			Cmd_RLen:=18;
			j:=(DelayAllarmeTemperaturaNonRaggiunta);   				(* Ritardo Allarme dall'avvio Caldaia*)
			TxLen:=TxLen+RAWTOHEX(ADR(j),2,ADR(TxData[TxLen]));
			j:=(DeltaInterventoAllarmeTempeaturaNonRaggiuta);			(* Delta Soglia Temperatura per Allarme Temperatura Non Raggiunta *)
			TxLen:=TxLen+RAWTOHEX(ADR(j),2,ADR(TxData[TxLen]));
			j:=(OffsetSetPointManuale);									(* Offest Perdite Scambiatore 1  *)
			TxLen:=TxLen+RAWTOHEX(ADR(j),2,ADR(TxData[TxLen]));
			j:=(OffsetSetPointManuale2);								(* Offest Perdite Scambiatore 2  *)
			TxLen:=TxLen+RAWTOHEX(ADR(j),2,ADR(TxData[TxLen]));
			j:=BOOL_TO_INT(BitAbilitaBoost);							(* Abilitazione controllo Boost  *)
			TxLen:=TxLen+RAWTOHEX(ADR(j),2,ADR(TxData[TxLen]));
			j:=BOOL_TO_INT(BitAbilitaBoost);										(* Offset al Setpoint della Caldaia per azione di Boost   *)
			TxLen:=TxLen+RAWTOHEX(ADR(j),2,ADR(TxData[TxLen]));




	6: (*  Scrivo i Parametri gestione Impianto - Antigelo   *)

			Cmd_Buf_U16:=ADR(Cmd_Buf[8]);
			SogliaMinStartAntigelo := Cmd_Buf_U16^; 			(* Soglia mininma Start Antigelo *)
			Cmd_Buf_U16:=ADR(Cmd_Buf[10]);
			SogliaMinStopAntigelo := Cmd_Buf_U16^;				(* Soglia Massima Stop Antigelo *)
			Cmd_Buf_U16:=ADR(Cmd_Buf[12]);
			BitAbilitaAntigelo :=INT_TO_BOOL( Cmd_Buf_U16^); 	(* Abilitazione Antigelo  *)

	7: (*  Leggi i parametri gestione Impianto - Antigelo *)

			Cmd_RLen:=14;
			j:=(SogliaMinStartAntigelo); 							(* Soglia mininma Start Antigelo *)
			TxLen:=TxLen+RAWTOHEX(ADR(j),2,ADR(TxData[TxLen]));
			j:=(SogliaMinStopAntigelo);								(* Soglia Massima Stop Antigelo *)
			TxLen:=TxLen+RAWTOHEX(ADR(j),2,ADR(TxData[TxLen]));
			j:=BOOL_TO_INT(BitAbilitaAntigelo);						(* Abilitazione Antigelo  *)
			TxLen:=TxLen+RAWTOHEX(ADR(j),2,ADR(TxData[TxLen]));

(*	10: (*  Scrivo i Parametri per la gestione della velocità dei circolatori sui primari   *)

			Cmd_Buf_U16:=ADR(Cmd_Buf[8]);
			PercVelMin := Cmd_Buf_U16^;
			Cmd_Buf_U16:=ADR(Cmd_Buf[10]);
			PercVelMax := Cmd_Buf_U16^;
			Cmd_Buf_U16:=ADR(Cmd_Buf[12]);
			ErroreTempMax := Cmd_Buf_U16^;
			Cmd_Buf_U16:=ADR(Cmd_Buf[14]);
			ErroreTempMin := Cmd_Buf_U16^;

	11: (*  Leggo i Parametri per la gestione della velocità dei circolatori sui primari   *)

			Cmd_RLen:=8;
			j:=(PercVelMin);
			TxLen:=TxLen+RAWTOHEX(ADR(j),2,ADR(TxData[TxLen]));
			j:=(PercVelMax);
			TxLen:=TxLen+RAWTOHEX(ADR(j),2,ADR(TxData[TxLen]));
			j:=(ErroreTempMax);
			TxLen:=TxLen+RAWTOHEX(ADR(j),2,ADR(TxData[TxLen]));
			j:=(ErroreTempMin);
			TxLen:=TxLen+RAWTOHEX(ADR(j),2,ADR(TxData[TxLen]));


	12: (*  Scrivo i Parametri per la gestione della velocità dei circolatori sui primari   *)


				Cmd_Buf_U16:=ADR(Cmd_Buf[8]);
				CAS01.DeltaTempThr := Cmd_Buf_U16^;
				Cmd_Buf_U16:=ADR(Cmd_Buf[10]);
				CAS01.Tmonitor_Off := DWORD_TO_TIME((Cmd_Buf_U16^)*60*1000);
				Cmd_Buf_U16:=ADR(Cmd_Buf[12]);
				CAS01.Tmonitor_On := DWORD_TO_TIME((Cmd_Buf_U16^)*60*1000);

	13: (*  Leggo i Parametri per la gestione della velocità dei circolatori sui primari   *)


				Cmd_RLen:=6;
				j:=(CAS01.DeltaTempThr);
				TxLen:=TxLen+RAWTOHEX(ADR(j),2,ADR(TxData[TxLen]));
				j:=DWORD_TO_WORD(TIME_TO_DWORD((CAS01.Tmonitor_Off)/60/1000));
				TxLen:=TxLen+RAWTOHEX(ADR(j),2,ADR(TxData[TxLen]));
				j:=DWORD_TO_WORD(TIME_TO_DWORD((CAS01.Tmonitor_On)/60/1000));
				TxLen:=TxLen+RAWTOHEX(ADR(j),2,ADR(TxData[TxLen]));


*)


	14: (*  Imposto data e ora del PLC  *)


			Cmd_Buf_U16:=ADR(Cmd_Buf[8]);
			SetAnno:= Cmd_Buf_U16^; 												(* Anno *)
			Cmd_Buf_U16:=ADR(Cmd_Buf[10]);
			SetMese:= Cmd_Buf_U16^;												 	(* mese *)
			Cmd_Buf_U16:=ADR(Cmd_Buf[12]);
			SetGiorno:=( Cmd_Buf_U16^);											 	(* Giorno *)
			Cmd_Buf_U16:=ADR(Cmd_Buf[14]);
			SetOra:=( Cmd_Buf_U16^); 												(* ora *)
			Cmd_Buf_U16:=ADR(Cmd_Buf[16]);
			SetMinuti:= ( Cmd_Buf_U16^);										 	(* Minuti *)
			Cmd_Buf_U16:=ADR(Cmd_Buf[18]);
			SetSecondi:= ( Cmd_Buf_U16^);										 	(* secondi *)

	(*		SysRtcSetTime(SetDataTime(DWORD_TO_INT(ADR(Cmd_Buf[8])),				(* Anno *)
										DWORD_TO_INT(ADR(Cmd_Buf[10])),				(* mese *)
										DWORD_TO_INT(ADR(Cmd_Buf[11])),				(* Giorno *)
										DWORD_TO_INT(ADR(Cmd_Buf[12])),				(* ora *)
										DWORD_TO_INT(ADR(Cmd_Buf[13])),				(* Minuti *)
										DWORD_TO_INT(ADR(Cmd_Buf[14]))				(* secondi *)
										)); *)

		SysRtcSetTime((SetDataTime(SetAnno,SetMese,SetGiorno,SetOra,SetMinuti,SetSecondi)));


ELSE
	Cmd_R:=3;
END_CASE
END_ACTION
ACTION Cmd_VAR:
(* Check index *)
IF Cmd_ObjIdx<1 OR  Cmd_ObjIdx>7   THEN
	Cmd_R:=2;
	RETURN;
END_IF

(* Process command *)

CASE Cmd_C OF

	1: (* SET Comandi  *)
		CASE Cmd_ObjIdx OF
			1:	Cmd_Buf_U16:=ADR(Cmd_Buf[8]);
				PLC_PRG.SelManAut := (Cmd_Buf_U16^);     (* Val 01 *)
				Cmd_Buf_U16:=ADR(Cmd_Buf[10]);
				PLC_PRG.SelC2_A_B :=(Cmd_Buf_U16^);	 (* Val 02 *)
				Cmd_Buf_U16:=ADR(Cmd_Buf[12]);
				PLC_PRG.SelC2B_INT := (Cmd_Buf_U16^);	 (* Val 03 *)
				Cmd_Buf_U16:=ADR(Cmd_Buf[14]);
				PLC_PRG.TGP_utente := (Cmd_Buf_U16^);	 (* Val 04 *)
				Cmd_Buf_U16:=ADR(Cmd_Buf[16]);
				PLC_PRG.TGP_min := (Cmd_Buf_U16^);	 	(* Val 05 *)
				Cmd_Buf_U16:=ADR(Cmd_Buf[18]);
				PLC_PRG.TGP_MAX := (Cmd_Buf_U16^);	 (* Val 06 *)
				Cmd_Buf_U16:=ADR(Cmd_Buf[20]);
				PLC_PRG.DEADZONE := (Cmd_Buf_U16^);			 (* Val 07 *)
				Cmd_Buf_U16:=ADR(Cmd_Buf[22]);
				DummyWord := (Cmd_Buf_U16^);	 		(* Val 08 *)
				Cmd_Buf_U16:=ADR(Cmd_Buf[24]);
				DummyWord := (Cmd_Buf_U16^);	 		(* Val 09 *)
				Cmd_Buf_U16:=ADR(Cmd_Buf[26]);
				DummyWord := (Cmd_Buf_U16^);	 		(* Val 10 *)



			2:	Cmd_Buf_U16:=ADR(Cmd_Buf[8]);
				PLC_PRG.TGP_203 := (Cmd_Buf_U16^);     (* Val 01 *)
				Cmd_Buf_U16:=ADR(Cmd_Buf[10]);
				PLC_PRG.TGP_303 :=(Cmd_Buf_U16^);	 	(* Val 02 *)
				Cmd_Buf_U16:=ADR(Cmd_Buf[12]);
				PLC_PRG.TGP_304 := (Cmd_Buf_U16^);	 	(* Val 03 *)
				Cmd_Buf_U16:=ADR(Cmd_Buf[14]);
				PLC_PRG.TGP_305 := (Cmd_Buf_U16^);	 	(* Val 04 *)
				Cmd_Buf_U16:=ADR(Cmd_Buf[16]);
				PLC_PRG.TGP_403 := (Cmd_Buf_U16^);	 	(* Val 05 *)
				Cmd_Buf_U16:=ADR(Cmd_Buf[18]);
				PLC_PRG.TGP_402 := (Cmd_Buf_U16^);	 	(* Val 06 *)
				Cmd_Buf_U16:=ADR(Cmd_Buf[20]);
				DummyWord := (Cmd_Buf_U16^);			 (* Val 07 *)
				Cmd_Buf_U16:=ADR(Cmd_Buf[22]);
				DummyWord := (Cmd_Buf_U16^);	 		(* Val 08 *)
				Cmd_Buf_U16:=ADR(Cmd_Buf[24]);
				DummyWord := (Cmd_Buf_U16^);	 		(* Val 09 *)
				Cmd_Buf_U16:=ADR(Cmd_Buf[26]);
				DummyWord := (Cmd_Buf_U16^);	 		(* Val 10 *)

			3:	Cmd_Buf_U16:=ADR(Cmd_Buf[8]);
				PLC_PRG.C2C_C101 := (Cmd_Buf_U16^);     (* Val 01 *)
				Cmd_Buf_U16:=ADR(Cmd_Buf[10]);
				PLC_PRG.C2C_C102 :=(Cmd_Buf_U16^);	 	(* Val 02 *)
				Cmd_Buf_U16:=ADR(Cmd_Buf[12]);
				PLC_PRG.C2C_C103 := (Cmd_Buf_U16^);	 	(* Val 03 *)
				Cmd_Buf_U16:=ADR(Cmd_Buf[14]);
				PLC_PRG.C2C_C104 := (Cmd_Buf_U16^);	 	(* Val 04 *)
				Cmd_Buf_U16:=ADR(Cmd_Buf[16]);
				PLC_PRG.C2C_C105 := (Cmd_Buf_U16^);	 	(* Val 05 *)
				Cmd_Buf_U16:=ADR(Cmd_Buf[18]);
				DummyWord:= (Cmd_Buf_U16^);	 	(* Val 06 *)
				Cmd_Buf_U16:=ADR(Cmd_Buf[20]);
				DummyWord := (Cmd_Buf_U16^);			 (* Val 07 *)
				Cmd_Buf_U16:=ADR(Cmd_Buf[22]);
				DummyWord  := (Cmd_Buf_U16^);	 		(* Val 08 *)
				Cmd_Buf_U16:=ADR(Cmd_Buf[24]);
				DummyWord  := (Cmd_Buf_U16^);	 		(* Val 09 *)
				Cmd_Buf_U16:=ADR(Cmd_Buf[26]);
				DummyWord  := (Cmd_Buf_U16^);	 		(* Val 10 *)

			4:	Cmd_Buf_U16:=ADR(Cmd_Buf[8]);
				PLC_PRG.DP_TGP_C101 := (Cmd_Buf_U16^);     (* Val 01 *)
				Cmd_Buf_U16:=ADR(Cmd_Buf[10]);
				PLC_PRG.DP_ASP_C101 :=(Cmd_Buf_U16^);	 	(* Val 02 *)
				Cmd_Buf_U16:=ADR(Cmd_Buf[12]);
				PLC_PRG.DP_OFP_C102 := (Cmd_Buf_U16^);	 	(* Val 03 *)
				Cmd_Buf_U16:=ADR(Cmd_Buf[14]);
				PLC_PRG.DP_TGP_C102 := (Cmd_Buf_U16^);	 	(* Val 04 *)
				Cmd_Buf_U16:=ADR(Cmd_Buf[16]);
				PLC_PRG.DP_OFP_C103 := (Cmd_Buf_U16^);	 	(* Val 05 *)
				Cmd_Buf_U16:=ADR(Cmd_Buf[18]);
				PLC_PRG.DP_TGP_C103 := (Cmd_Buf_U16^);	 	(* Val 06 *)
				Cmd_Buf_U16:=ADR(Cmd_Buf[20]);
				PLC_PRG.DP_OFP_C104  := (Cmd_Buf_U16^);			 (* Val 07 *)
				Cmd_Buf_U16:=ADR(Cmd_Buf[22]);
				PLC_PRG.DP_TGP_C104  := (Cmd_Buf_U16^);	 		(* Val 08 *)
				Cmd_Buf_U16:=ADR(Cmd_Buf[24]);
				PLC_PRG.DP_TGP_C105  := (Cmd_Buf_U16^);	 		(* Val 09 *)
				Cmd_Buf_U16:=ADR(Cmd_Buf[26]);
				PLC_PRG.DP_ASP_C105  := (Cmd_Buf_U16^);	 		(* Val 10 *)


			5:	Cmd_Buf_U16:=ADR(Cmd_Buf[8]);
				DummyWord := (Cmd_Buf_U16^);     (* Val 01 *)
				Cmd_Buf_U16:=ADR(Cmd_Buf[10]);
				DummyWord :=(Cmd_Buf_U16^);	 	(* Val 02 *)
				Cmd_Buf_U16:=ADR(Cmd_Buf[12]);
				DummyWord := (Cmd_Buf_U16^);	 	(* Val 03 *)
				Cmd_Buf_U16:=ADR(Cmd_Buf[14]);
				DummyWord := (Cmd_Buf_U16^);	 	(* Val 04 *)
				Cmd_Buf_U16:=ADR(Cmd_Buf[16]);
				DummyWord := (Cmd_Buf_U16^);	 	(* Val 05 *)
				Cmd_Buf_U16:=ADR(Cmd_Buf[18]);
				DummyWord := (Cmd_Buf_U16^);	 	(* Val 06 *)
				Cmd_Buf_U16:=ADR(Cmd_Buf[20]);
				DummyWord  := (Cmd_Buf_U16^);			 (* Val 07 *)
				Cmd_Buf_U16:=ADR(Cmd_Buf[22]);
				DummyWord  := (Cmd_Buf_U16^);	 		(* Val 08 *)
				Cmd_Buf_U16:=ADR(Cmd_Buf[24]);
				DummyWord  := (Cmd_Buf_U16^);	 		(* Val 09 *)
				Cmd_Buf_U16:=ADR(Cmd_Buf[26]);
				DummyWord  := (Cmd_Buf_U16^);	 		(* Val 10 *)

			6:	Cmd_Buf_U16:=ADR(Cmd_Buf[8]);
				DummyWord := (Cmd_Buf_U16^);     (* Val 01 *)
				Cmd_Buf_U16:=ADR(Cmd_Buf[10]);
				DummyWord :=(Cmd_Buf_U16^);	 	(* Val 02 *)
				Cmd_Buf_U16:=ADR(Cmd_Buf[12]);
				DummyWord := (Cmd_Buf_U16^);	 	(* Val 03 *)
				Cmd_Buf_U16:=ADR(Cmd_Buf[14]);
				DummyWord := (Cmd_Buf_U16^);	 	(* Val 04 *)
				Cmd_Buf_U16:=ADR(Cmd_Buf[16]);
				DummyWord := (Cmd_Buf_U16^);	 	(* Val 05 *)
				Cmd_Buf_U16:=ADR(Cmd_Buf[18]);
				DummyWord := (Cmd_Buf_U16^);	 	(* Val 06 *)
				Cmd_Buf_U16:=ADR(Cmd_Buf[20]);
				DummyWord  := (Cmd_Buf_U16^);			 (* Val 07 *)
				Cmd_Buf_U16:=ADR(Cmd_Buf[22]);
				DummyWord  := (Cmd_Buf_U16^);	 		(* Val 08 *)
				Cmd_Buf_U16:=ADR(Cmd_Buf[24]);
				DummyWord  := (Cmd_Buf_U16^);	 		(* Val 09 *)
				Cmd_Buf_U16:=ADR(Cmd_Buf[26]);
				DummyWord  := (Cmd_Buf_U16^);	 		(* Val 10 *)

			7:	Cmd_Buf_U16:=ADR(Cmd_Buf[8]);
				DummyWord := (Cmd_Buf_U16^);     (* Val 01 *)
				Cmd_Buf_U16:=ADR(Cmd_Buf[10]);
				DummyWord :=(Cmd_Buf_U16^);	 	(* Val 02 *)
				Cmd_Buf_U16:=ADR(Cmd_Buf[12]);
				DummyWord := (Cmd_Buf_U16^);	 	(* Val 03 *)
				Cmd_Buf_U16:=ADR(Cmd_Buf[14]);
				DummyWord := (Cmd_Buf_U16^);	 	(* Val 04 *)
				Cmd_Buf_U16:=ADR(Cmd_Buf[16]);
				DummyWord := (Cmd_Buf_U16^);	 	(* Val 05 *)
				Cmd_Buf_U16:=ADR(Cmd_Buf[18]);
				DummyWord := (Cmd_Buf_U16^);	 	(* Val 06 *)
				Cmd_Buf_U16:=ADR(Cmd_Buf[20]);
				DummyWord  := (Cmd_Buf_U16^);			 (* Val 07 *)
				Cmd_Buf_U16:=ADR(Cmd_Buf[22]);
				DummyWord  := (Cmd_Buf_U16^);	 		(* Val 08 *)
				Cmd_Buf_U16:=ADR(Cmd_Buf[24]);
				DummyWord  := (Cmd_Buf_U16^);	 		(* Val 09 *)
				Cmd_Buf_U16:=ADR(Cmd_Buf[26]);
				DummyWord  := (Cmd_Buf_U16^);	 		(* Val 10 *)


		END_CASE


	2: (* GET Comandi  *)
		CASE Cmd_ObjIdx OF

			1: (*  Leggi i parametri gestione Impianto  *)
			Cmd_RLen:=10;
			j:=(PLC_PRG.SelManAut);
			TxLen:=TxLen+RAWTOHEX(ADR(j),2,ADR(TxData[TxLen]));
			j:=(PLC_PRG.SelC2_A_B);
			TxLen:=TxLen+RAWTOHEX(ADR(j),2,ADR(TxData[TxLen]));
			j:=(PLC_PRG.SelC2B_INT);
			TxLen:=TxLen+RAWTOHEX(ADR(j),2,ADR(TxData[TxLen]));
			j:=(PLC_PRG.TGP_utente);
			TxLen:=TxLen+RAWTOHEX(ADR(j),2,ADR(TxData[TxLen]));
			j:=(PLC_PRG.TGP_min);
			TxLen:=TxLen+RAWTOHEX(ADR(j),2,ADR(TxData[TxLen]));
			j:=(PLC_PRG.TGP_MAX);
			TxLen:=TxLen+RAWTOHEX(ADR(j),2,ADR(TxData[TxLen]));
			j:=(PLC_PRG.DEADZONE);
			TxLen:=TxLen+RAWTOHEX(ADR(j),2,ADR(TxData[TxLen]));
			j:=(0);
			TxLen:=TxLen+RAWTOHEX(ADR(j),2,ADR(TxData[TxLen]));
			j:=(0);
			TxLen:=TxLen+RAWTOHEX(ADR(j),2,ADR(TxData[TxLen]));
			j:=(0);
			TxLen:=TxLen+RAWTOHEX(ADR(j),2,ADR(TxData[TxLen]));

			2: (*  Leggi i parametri gestione Impianto  *)
			Cmd_RLen:=10;
			j:=(PLC_PRG.TGP_203);
			TxLen:=TxLen+RAWTOHEX(ADR(j),2,ADR(TxData[TxLen]));
			j:=(PLC_PRG.TGP_303);
			TxLen:=TxLen+RAWTOHEX(ADR(j),2,ADR(TxData[TxLen]));
			j:=(PLC_PRG.TGP_304);
			TxLen:=TxLen+RAWTOHEX(ADR(j),2,ADR(TxData[TxLen]));
			j:=(PLC_PRG.TGP_305);
			TxLen:=TxLen+RAWTOHEX(ADR(j),2,ADR(TxData[TxLen]));
			j:=(PLC_PRG.TGP_403);
			TxLen:=TxLen+RAWTOHEX(ADR(j),2,ADR(TxData[TxLen]));
			j:=(PLC_PRG.TGP_402);
			TxLen:=TxLen+RAWTOHEX(ADR(j),2,ADR(TxData[TxLen]));
			j:=(0);
			TxLen:=TxLen+RAWTOHEX(ADR(j),2,ADR(TxData[TxLen]));
			j:=(0);
			TxLen:=TxLen+RAWTOHEX(ADR(j),2,ADR(TxData[TxLen]));
			j:=(0);
			TxLen:=TxLen+RAWTOHEX(ADR(j),2,ADR(TxData[TxLen]));
			j:=(0);
			TxLen:=TxLen+RAWTOHEX(ADR(j),2,ADR(TxData[TxLen]));

			3: (*  Leggi i parametri gestione Impianto  *)
			Cmd_RLen:=10;
			j:=(PLC_PRG.C2C_C101);
			TxLen:=TxLen+RAWTOHEX(ADR(j),2,ADR(TxData[TxLen]));
			j:=(PLC_PRG.C2C_C102);
			TxLen:=TxLen+RAWTOHEX(ADR(j),2,ADR(TxData[TxLen]));
			j:=(PLC_PRG.C2C_C103);
			TxLen:=TxLen+RAWTOHEX(ADR(j),2,ADR(TxData[TxLen]));
			j:=(PLC_PRG.C2C_C104);
			TxLen:=TxLen+RAWTOHEX(ADR(j),2,ADR(TxData[TxLen]));
			j:=(PLC_PRG.C2C_C105);
			TxLen:=TxLen+RAWTOHEX(ADR(j),2,ADR(TxData[TxLen]));
			j:=(COMPRESSORE01.MB_RegistriHoldingLetti[3]);
			TxLen:=TxLen+RAWTOHEX(ADR(j),2,ADR(TxData[TxLen]));
			j:=(COMPRESSORE02.MB_RegistriHoldingLetti[3]);
			TxLen:=TxLen+RAWTOHEX(ADR(j),2,ADR(TxData[TxLen]));
			j:=(COMPRESSORE03.MB_RegistriHoldingLetti[3]);
			TxLen:=TxLen+RAWTOHEX(ADR(j),2,ADR(TxData[TxLen]));
			j:=(COMPRESSORE04.MB_RegistriHoldingLetti[3]);
			TxLen:=TxLen+RAWTOHEX(ADR(j),2,ADR(TxData[TxLen]));
			j:=(COMPRESSORE05.MB_RegistriHoldingLetti[3]);
			TxLen:=TxLen+RAWTOHEX(ADR(j),2,ADR(TxData[TxLen]));

			4: (*  Leggi i parametri gestione Impianto  *)
			Cmd_RLen:=10;
			j:=(PLC_PRG.DP_TGP_C101);
			TxLen:=TxLen+RAWTOHEX(ADR(j),2,ADR(TxData[TxLen]));
			j:=(PLC_PRG.DP_ASP_C101);
			TxLen:=TxLen+RAWTOHEX(ADR(j),2,ADR(TxData[TxLen]));
			j:=(PLC_PRG.DP_OFP_C102);
			TxLen:=TxLen+RAWTOHEX(ADR(j),2,ADR(TxData[TxLen]));
			j:=(PLC_PRG.DP_TGP_C102);
			TxLen:=TxLen+RAWTOHEX(ADR(j),2,ADR(TxData[TxLen]));
			j:=(PLC_PRG.DP_OFP_C103);
			TxLen:=TxLen+RAWTOHEX(ADR(j),2,ADR(TxData[TxLen]));
			j:=(PLC_PRG.DP_TGP_C103);
			TxLen:=TxLen+RAWTOHEX(ADR(j),2,ADR(TxData[TxLen]));
			j:=(PLC_PRG.DP_OFP_C104);
			TxLen:=TxLen+RAWTOHEX(ADR(j),2,ADR(TxData[TxLen]));
			j:=(PLC_PRG.DP_TGP_C104);
			TxLen:=TxLen+RAWTOHEX(ADR(j),2,ADR(TxData[TxLen]));
			j:=(PLC_PRG.DP_TGP_C105);
			TxLen:=TxLen+RAWTOHEX(ADR(j),2,ADR(TxData[TxLen]));
			j:=(PLC_PRG.DP_ASP_C105);
			TxLen:=TxLen+RAWTOHEX(ADR(j),2,ADR(TxData[TxLen]));

			5: (*  Leggi i parametri gestione Impianto  *)
			Cmd_RLen:=10;
			j:=(SEL(PX01.ERR,px01.ValoreScalato,FPT01.IntPressioneCalcolata));
			TxLen:=TxLen+RAWTOHEX(ADR(j),2,ADR(TxData[TxLen]));
			j:=(PLC_PRG.DP_C2A);
			TxLen:=TxLen+RAWTOHEX(ADR(j),2,ADR(TxData[TxLen]));
			j:=(PLC_PRG.DP_C2B);
			TxLen:=TxLen+RAWTOHEX(ADR(j),2,ADR(TxData[TxLen]));
			j:=(SEL((FPT06.Status_Log=0),9999,DWORD_TO_INT(FPT06.IntPressioneCalcolata)));
			TxLen:=TxLen+RAWTOHEX(ADR(j),2,ADR(TxData[TxLen]));
			j:=(SEL((FPT07.Status_Log=0),9999,DWORD_TO_INT(FPT07.IntPressioneCalcolata)));
			TxLen:=TxLen+RAWTOHEX(ADR(j),2,ADR(TxData[TxLen]));
			j:=(SEL((FPT08.Status_Log=0),9999,DWORD_TO_INT(FPT08.IntPressioneCalcolata)));
			TxLen:=TxLen+RAWTOHEX(ADR(j),2,ADR(TxData[TxLen]));
			j:=(SEL((FPT09.Status_Log=0),9999,DWORD_TO_INT(FPT09.IntPressioneCalcolata)));
			TxLen:=TxLen+RAWTOHEX(ADR(j),2,ADR(TxData[TxLen]));
			j:=(SEL((FPT10.Status_Log=0),9999,DWORD_TO_INT(FPT10.IntPressioneCalcolata)));
			TxLen:=TxLen+RAWTOHEX(ADR(j),2,ADR(TxData[TxLen]));
			j:=(SEL((FPT05.Status_Log=0),9999,DWORD_TO_INT(FPT05.IntPressioneCalcolata)));
			TxLen:=TxLen+RAWTOHEX(ADR(j),2,ADR(TxData[TxLen]));
			j:=(0);
			TxLen:=TxLen+RAWTOHEX(ADR(j),2,ADR(TxData[TxLen]));

			6: (*  Leggi i parametri gestione Impianto  *)
			Cmd_RLen:=10;
			j:=(PLC_PRG.TGP_C101);
			(*j:=COMPRESSORE01.MB_RegistriHoldingLetti[112] *)
			TxLen:=TxLen+RAWTOHEX(ADR(j),2,ADR(TxData[TxLen]));
			j:=(PLC_PRG.ASP_C101);
			TxLen:=TxLen+RAWTOHEX(ADR(j),2,ADR(TxData[TxLen]));
			j:=(PLC_PRG.ONP_C102);
			TxLen:=TxLen+RAWTOHEX(ADR(j),2,ADR(TxData[TxLen]));
			j:=(PLC_PRG.OFP_C102);
			TxLen:=TxLen+RAWTOHEX(ADR(j),2,ADR(TxData[TxLen]));
			j:=(PLC_PRG.ONP_C103);
			TxLen:=TxLen+RAWTOHEX(ADR(j),2,ADR(TxData[TxLen]));
			j:=(PLC_PRG.OFP_C103);
			TxLen:=TxLen+RAWTOHEX(ADR(j),2,ADR(TxData[TxLen]));
			j:=(PLC_PRG.ONP_C104);
			TxLen:=TxLen+RAWTOHEX(ADR(j),2,ADR(TxData[TxLen]));
			j:=(PLC_PRG.OFP_C104);
			TxLen:=TxLen+RAWTOHEX(ADR(j),2,ADR(TxData[TxLen]));
			j:=(PLC_PRG.TGP_C105);
			TxLen:=TxLen+RAWTOHEX(ADR(j),2,ADR(TxData[TxLen]));
			j:=(PLC_PRG.ASP_C105);
			TxLen:=TxLen+RAWTOHEX(ADR(j),2,ADR(TxData[TxLen]));

			7: (*  Leggi i parametri gestione Impianto  *)
			Cmd_RLen:=10;
			j:=COMPRESSORE01.MB_RegistriHoldingLetti[112];
			TxLen:=TxLen+RAWTOHEX(ADR(j),2,ADR(TxData[TxLen]));
			j:=COMPRESSORE01.MB_RegistriHoldingLetti[113];
			TxLen:=TxLen+RAWTOHEX(ADR(j),2,ADR(TxData[TxLen]));
			j:=COMPRESSORE02.MB_RegistriHoldingLetti[113];
			TxLen:=TxLen+RAWTOHEX(ADR(j),2,ADR(TxData[TxLen]));
			j:=COMPRESSORE02.MB_RegistriHoldingLetti[112];
			TxLen:=TxLen+RAWTOHEX(ADR(j),2,ADR(TxData[TxLen]));
			j:=COMPRESSORE03.MB_RegistriHoldingLetti[113];
			TxLen:=TxLen+RAWTOHEX(ADR(j),2,ADR(TxData[TxLen]));
			j:=COMPRESSORE03.MB_RegistriHoldingLetti[112];
			TxLen:=TxLen+RAWTOHEX(ADR(j),2,ADR(TxData[TxLen]));
			j:=COMPRESSORE04.MB_RegistriHoldingLetti[113];
			TxLen:=TxLen+RAWTOHEX(ADR(j),2,ADR(TxData[TxLen]));
			j:=COMPRESSORE04.MB_RegistriHoldingLetti[112];
			TxLen:=TxLen+RAWTOHEX(ADR(j),2,ADR(TxData[TxLen]));
			j:=COMPRESSORE05.MB_RegistriHoldingLetti[112];
			TxLen:=TxLen+RAWTOHEX(ADR(j),2,ADR(TxData[TxLen]));
			j:=COMPRESSORE05.MB_RegistriHoldingLetti[113];
			TxLen:=TxLen+RAWTOHEX(ADR(j),2,ADR(TxData[TxLen]));







		END_CASE

ELSE
	Cmd_R:=3;
END_CASE
END_ACTION
ACTION Command:
(* Default response OK/NODATA *)
Cmd_R:=0;
Cmd_RLen:=0;
TxLen:=16;

(* Check object *)
CASE Cmd_Obj OF

	EO_SYS:
		Cmd_SYS();

	EO_COMPINGRR:
		Cmd_COMPINGRR();

	EO_COMPINGRML:
		Cmd_COMPINGRML();

	EO_VAR:
		Cmd_VAR();

ELSE
	Cmd_R:=1;
END_CASE

(* Generate response *)
IF TxLen>0 THEN
	RAWTOHEX(ADR(Cmd_Obj)	,2,ADR(TxData[ 0]));
	RAWTOHEX(ADR(Cmd_ObjIdx),2,ADR(TxData[ 4]));
	RAWTOHEX(ADR(Cmd_R)		,2,ADR(TxData[ 8]));
	RAWTOHEX(ADR(Cmd_RLen)	,2,ADR(TxData[12]));
	TxTrig:=TRUE;
END_IF
END_ACTION

(* POU Utils Functions/TCPSERVER, ST *)
FUNCTION_BLOCK TCPSERVER
(***********************************************************************************************************	*)
(* Version: 1.6                                    			          											*)
(* Date: 11.02.2011                                   					          							    *)
(***********************************************************************************************************	*)
(* WAGO Kontakttechnik GmbH Hansastr. 27 32423 Minden(Westf.)													*)
(* Tel. +0049 571/887-0 Fax. +0049 571/887-0																	*)
(* Author: VB																									*)
(***********************************************************************************************************	*)
(*Description:	A TCP server to read and write data													       		*)
(*Historie:																										*)
(*Version 1.6: 11.02.2011: Changes according to 750-880/881											 			*)
(*Version 1.5: 27.11.2008 Bugfix allow reuse port																*)
(*Version 1.4: 13.10.2008 Bugfix transmitting large data														*)
(*Version 1.3: 15.01.2007 Changes according to FW11																*)
(*Version 1.2: 09.03.2006 Changes for socket handle 0											       			*)
(*Version 1.1: 14.02.2005 Release																				*)
(***********************************************************************************************************	*)
VAR CONSTANT
	STATE_INIT     				 : BYTE:= 0;
	STATE_OPEN     				 : BYTE:= 1;
	STATE_TX       				 : BYTE:= 20;
	STATE_RX       				 : BYTE:= 30;
	STATE_CLOSE    				 : BYTE:= 40;
	STATE_ERROR_TRAP		 	 : BYTE:= 200;
END_VAR
VAR_INPUT
	xEnable    					: BOOL;	 (* Set TRUE to enable function block *)
	wPortNumber					: WORD;  (* Port *)
	tServerTimeOut				: TIME:=t#50s;
	ptSendData					: POINTER TO ARRAY[0..MAX_SEND_TCP_SERVER] OF BYTE;
	diSendCount					: DINT;
END_VAR
VAR_OUTPUT
	xClientConnected  			: BOOL:= FALSE;
	diError 					: DINT:= 0;
END_VAR
(* Status Codes -----------------------------------------
	16#8001 => No socket descriptor available 
	16#8002 => SysSockBind fails 
	16#8003 => SysSockListen fails 
	16#8004 => switching to none blocking mode fails
	16#8005 => SysSockClose() returns FALSE 
    16#8006 => SysSockConnect() fails
    16#8007 => SysSockSend() fails
	16#8008 => error state machine 
	16#8009 => timeout while waiting for data from server 
	16#0001 => server waiting for client to establish connection
------------------------------------------------------------*)
VAR_IN_OUT
	xStartSend					: BOOL;
	aReceiveBuffer				: ARRAY [0..MAX_RECEIVE_TCP_SERVER] OF BYTE;
	diReceiveCount				: DINT;
END_VAR

VAR
	m_State    					: BYTE:= 0;
	m_ReceiveBuffer				: ARRAY [0..MAX_RECEIVE_TCP_SERVER_SOCKET] OF BYTE;
	m_ServerSocket				: DINT:= SOCKET_INVALID;
	m_Socket					: DINT:= SOCKET_INVALID;
	m_AddressInfo				: SOCKADDRESS;
	m_BytesReceived				: DINT;
	m_diReturn					: DINT;
	m_xReturn					: BOOL;
	m_SizeSockadr				: DWORD;
	m_ConnectionWatchdog		: TON;
	m_Flags						: DINT;
	m_NoneBlocking   			: DINT:= 1;
	m_Blocking   				: DINT:= 0;
	i							: INT;
	m_count						: DINT;
	diOption					: DINT := 1;
	on: DINT;
END_VAR
IF xEnable THEN
	CASE m_State OF
		STATE_INIT:
			(* Create Socket *)
			m_ServerSocket:= SysSockCreate( SOCKET_AF_INET, SOCKET_STREAM, 0);
			IF m_ServerSocket = SOCKET_INVALID THEN
				(* *)
				diError:= 16#8001;
				m_State:= STATE_ERROR_TRAP;
				RETURN;
			ELSE
				;
			END_IF
			(* Address bindings *)
			(********************)
			on:=1;
			SysSockSetOption( m_ServerSocket, SOCKET_SOL, SOCKET_SO_REUSEADDR, ADR(on), SIZEOF(on) );

			m_AddressInfo.sin_family:= SOCKET_AF_INET;
			m_AddressInfo.sin_port  := SysSockHtons( wPortNumber);
			m_AddressInfo.sin_addr  := SOCKET_INADDR_ANY;
			IF NOT SysSockBind( m_ServerSocket, ADR(m_AddressInfo), SIZEOF(m_AddressInfo)) THEN
				diError:= 16#8002;
				m_State:= STATE_ERROR_TRAP;
				RETURN;
			END_IF
			(* Wait for connections *)
			(************************)
			IF NOT SysSockListen( m_ServerSocket, 1) THEN
				diError:= 16#8003;
				m_State:= STATE_ERROR_TRAP;
			END_IF

			(* Puts SOCKET in NonBlocking mode *)
			m_diReturn:= SysSockIoctl( m_ServerSocket, SOCKET_FIONBIO, ADR(m_NoneBlocking));

			m_State:= STATE_OPEN;


		STATE_OPEN: 	(* Waiting for incomming connection *)
				m_SizeSockadr:=SIZEOF(m_AddressInfo);
				m_Socket:= SysSockAccept( m_ServerSocket, ADR(m_AddressInfo), ADR(m_SizeSockadr));
				diError:=State_open;
				IF m_Socket <> SOCKET_INVALID THEN
					xClientConnected:=TRUE;
					(*Set Push-Bit:new V1.5*)
					IF ADR(%MW0)=16#30000000  OR ADR(%MW0)=16#20000000 THEN (*841 or 881*)
						SysSockSetOption(
							diSocket:=m_Socket,
							diLevel:=6,
							diOption:=SOCKET_TCP_NODELAY,
							pOptionValue:=ADR(diOption),
							diOptionLength:=SIZEOF(diOption));
					ELSE
							;
					END_IF
					SysSockIoctl( m_Socket, SOCKET_FIONBIO, ADR(m_NoneBlocking));
					m_State:= STATE_RX;
					diError:=0;
				END_IF

		STATE_RX:
					m_BytesReceived:= SysSockRecv( m_Socket, ADR(m_ReceiveBuffer), SIZEOF(m_ReceiveBuffer), 0);
					CASE m_BytesReceived OF
					-1:(*no data available or error occured*)
						m_ConnectionWatchdog(IN:=TRUE , PT:=tServerTimeOut );
						IF m_connectionWatchdog.Q THEN
							m_State:= STATE_CLOSE;
							m_ConnectionWatchdog(IN:=FALSE);(*reset connection watchdog*)
							diError := 16#8009;
						END_IF
					0:(* socket was "gracefully closed"  *)
						m_State:= STATE_CLOSE;
						diError := 16#8003;
					ELSE
						(* Copy received data into receive buffer *)
						(********************************)
						FOR i:= 0 TO DINT_TO_INT(m_BytesReceived	)-1 DO
							aReceiveBuffer[diReceiveCount]:= m_ReceiveBuffer[i];
							diReceiveCount:=(diReceiveCount+1) MOD SIZEOF(aReceiveBuffer);
						END_FOR

						m_ConnectionWatchdog(IN:=FALSE);(*reset connection watchdog*)
					END_CASE

				(*send data*)
				IF xStartSend	 THEN
					m_State := STATE_TX;
				END_IF

	STATE_TX:	 (* send TCP-message *)
		m_diReturn := SysSockSend(diSocket := m_Socket,
								  pbyBuffer := ADR(ptSendData^[m_count]),(*geändert V1.4 bisher: [0] *)
								  diBufferSize := diSendCount-m_count,
								  diFlags :=m_Flags);
		CASE m_diReturn OF
		-1:	(* ERROR or data could not yet be send (V1.3 due to new FW11) *)
			m_ConnectionWatchdog(IN:=TRUE , PT:=tServerTimeOut );
			IF m_connectionWatchdog.Q THEN
				m_State:= STATE_CLOSE;
				m_ConnectionWatchdog(IN:=FALSE);(*reset connection watchdog*)
				diError := 16#8007;
			END_IF
		0: (* socket was "gracefully closed"  *)
			m_State := STATE_CLOSE;
			diError := 16#8003;
		ELSE (* succesful *)
			m_count:=m_count+m_diReturn;
			IF m_count>=diSendCount THEN
				diError := 16#0000;
				m_State := STATE_RX;
				m_count:=0;
				xStartSend:=FALSE;
			END_IF
			m_ConnectionWatchdog(IN:=FALSE);(*reset connection watchdog*)
		END_CASE


		STATE_CLOSE:	(* Close the server *)

		IF ADR(%MW0)=16#30000000  OR ADR(%MW0)=16#20000000 THEN (*841 or 881*)
			;
		ELSE
			IF m_Socket>=0 THEN
				SysSockShutdown(m_Socket, 0);;(*870*)
			END_IF
		END_IF
		IF m_Socket>=0 THEN
			SysSockClose( m_Socket);
		END_IF
		xClientConnected:= FALSE;
		m_State:= STATE_OPEN; (* Try to open the server again *)
		m_ConnectionWatchdog(IN:=FALSE);(*reset connection watchdog*)

		STATE_ERROR_TRAP: (* Error Read/Write socket  *)
			m_State:= STATE_ERROR_TRAP;

	ELSE  (* Bad FSM code trap  *)
			m_State:= STATE_ERROR_TRAP;
			diError:= 16#8008;
	END_CASE;
ELSE
	IF m_State <> STATE_INIT THEN
		IF ADR(%MW0)=16#30000000  OR ADR(%MW0)=16#20000000 THEN (*841 or 881*)
			;
		ELSE
			IF m_Socket>=0 THEN
				SysSockShutdown(m_Socket, 0);;(*870*)
			END_IF
		END_IF
		IF m_Socket>=0 THEN
			SysSockClose( m_Socket);
		END_IF
		IF ADR(%MW0)=16#30000000  OR ADR(%MW0)=16#20000000 THEN (*841 or 881*)
			;
		ELSE
			IF m_ServerSocket>=0 THEN
				SysSockShutdown(m_ServerSocket, 0);;(*870*)
			END_IF
		END_IF
		IF m_ServerSocket>=0 THEN
			SysSockClose( m_ServerSocket);
		END_IF
		xClientConnected:= FALSE;
		diError:= 0;
		m_State:= STATE_init; (* Try to open the server again *)
		m_ConnectionWatchdog(IN:=FALSE);(*reset connection watchdog*)
	END_IF
END_IF
END_FUNCTION_BLOCK

(* POU Utils Functions/HEXTORAW, ST *)
FUNCTION HEXTORAW : WORD
VAR_INPUT
	pString		: POINTER TO BYTE;
	StringLen	: WORD;
	pData		: POINTER TO BYTE;
END_VAR
VAR
	xl: WORD;
	xi: WORD;
	xr: BYTE;
END_VAR
xl:=0;
xi:=0;

WHILE xi<StringLen DO

	IF pString^>=97 AND pString^<=102 THEN
		xr := pString^ - 87;
	ELSIF pString^>=65 AND pString^<=70 THEN
		xr := pString^ - 55;
	ELSIF pString^>=48 AND pString^<=57 THEN
		xr := pString^ - 48;
	ELSE
		xr := 16;
	END_IF

	IF xr<16 THEN
		IF (xi AND 1)=0 THEN
			pData^ := xr * 16;
		ELSE
			pData^ := pData^ + xr;
			pData := pData + 1;
			xl := xl + 1;
		END_IF
	END_IF

	xi := xi + 1;
	pString := pString + 1;

END_WHILE

HEXTORAW:=xl;
END_FUNCTION

(* POU TCP_Remote/LogTrig, ST *)
FUNCTION LogTrig : BOOL
VAR
	s1 : STRING(160);
	i  : BYTE;
	j  : WORD;
	BitTest: BOOL;
END_VAR
BitTest:=TRUE;

(*

(*---------------------------------------------------------------*)
	Logger_Head();
(*---------------------------------------------------------------*)

PX01.AddLogData();
PX02.AddLogData();
PX03.AddLogData();
PX04.AddLogData();
Logger_Send();


Logger_Head();

(*
FOR i:=1 TO Plant_ANZ_INEPRO DO
	ANZ_INEPRO[i].AddLogData();
END_FOR *)
ANZ_INEPRO[1].AddLogData();
ANZ_INEPRO[2].AddLogData();
Logger_Send();


Logger_Head();

ANZ_INEPRO[3].AddLogData();
ANZ_INEPRO[4].AddLogData();
Logger_Send();


Logger_Head();
ANZ_INEPRO[5].AddLogData();

Logger_Send();


Logger_Head();

	COMPRESSORE01.AddLogData(ModBus:=MODB02);
	COMPRESSORE05.AddLogData(ModBus:=MODB02);
Logger_Send();


Logger_Head();
	COMPRESSORE02.AddLogData(ModBus:=MODB03);
	COMPRESSORE03.AddLogData(ModBus:=MODB03);
	COMPRESSORE04.AddLogData(ModBus:=MODB03);
Logger_Send();


Logger_Head();

	FPT01.AddLogData(ModBus:=MODB05);
	FPT02.AddLogData();
	FPT03.AddLogData();
	FPT04.AddLogData();
	FPT05.AddLogData();
	FPT06.AddLogData();
	FPT07.AddLogData();
	FPT08.AddLogData();
	FPT09.AddLogData();
	FPT10.AddLogData();

(*	ESSICATORE01.AddLogData(ModBus:=MODB04); *)
(*	ESSICATORE02.AddLogData(ModBus:=MODB04); *)



(*---------------------------------------------------------------*)
	Logger_Send();
(*---------------------------------------------------------------*)
*)
END_FUNCTION

(* POU Utils Functions/RAWTOHEX, ST *)
FUNCTION RAWTOHEX : WORD
VAR_INPUT
	pData: POINTER TO BYTE;
	DataLen: WORD;
	pString: POINTER TO BYTE;
END_VAR
VAR
	xl: WORD;
END_VAR
xl:=0;

WHILE DataLen>0 DO

	pString^ := (pData^ / 16#10) + 48 + (((pData^ / 16#10)/10)*7);
	pString:=pString+1;
	pString^ := (pData^ AND 16#0F)  + 48 + (((pData^ AND 16#0F)/10)*7);
	pString:=pString+1;
	pData:=pData+1;
	DataLen:=DataLen-1;
	xl:=xl+2;

END_WHILE

(*pString^:=0;*)

RAWTOHEX:=xl;
END_FUNCTION

(* POU Utils Functions/GestioneDataTime_DaOscat/SetDataTime, ST *)
FUNCTION SetDataTime : DT
VAR_INPUT
	year : INT;
	month : INT;
	day : INT;
	hour : INT;
	minute : INT;
	second : INT;
END_VAR

VAR
	count : INT;
END_VAR
(* Creazione variabiletipo DT per creare Orario da dare al PLC *)


IF month > 2 THEN
	count := (month - 1) * 30;
	IF month > 7 THEN count := count + SHR(month - 3,1); ELSE count := count + SHR(month - 4,1); END_IF;
	(* chech for leap year and add one day if true *)
	IF SHL(year,14) = 0 THEN count := count + 1; END_IF;
ELSE
	count := (month - 1) * 31;
END_IF;


SetDataTime := DWORD_TO_DT(DATE_TO_DWORD( DWORD_TO_DATE((INT_TO_DWORD(count + day - 1) + SHR(INT_TO_DWORD(year) * 1461 - 2878169, 2)) * 86400))
				+ INT_TO_DWORD(SECOND)
				+ INT_TO_DWORD(MINUTE) * 60
				+ INT_TO_DWORD(HOUR) * 3600);
END_FUNCTION

(* POU Plant/SYS_Proc, ST *)
PROGRAM SYS_Proc
VAR
	fALARM_PB		:FLT_TAP;
	fALARM_TB		:FLT_TAP;
	fALARM_PM		:FLT_TAP;
	fALARM_ALARM_PM_PB_TB		:FLT_TAP;

(*	fGZB_ST			:FLT_TAP;  (* GATEWAY ZIGBEE *)*)
	fVPN_ST1		:FLT_TAP;  (* VPN CONNECT *)
	fVPN_ST2		:FLT_TAP;  (* VPN STATUS *)
	fKEY_CT_ST		:FLT_TAP;  (* DOOR1 *)
	fKEY_SCT_ST		:FLT_TAP;  (* DOOR2 *)
	fKEY_QE_ST		:FLT_TAP;  (* DOOR3 *)


	fBostAttivo	:FLT_TAP;

	fALARM_MancatoRaggiungimentoAcqua		:FLT_TAP;
	DelayfALARM_MancatoRaggiungimentoAcqua:TON;

END_VAR
(*************** ISPESL *****************)
(*
fALARM_PB(IN:=ALARM_PB);
IF fALARM_PB.EVH THEN
	LogEv(EL_AlarmStop,EO_PBV,1,1,'Over_Pressure_Alarm');
END_IF

fALARM_TB(IN:=ALARM_TB);
IF fALARM_TB.EVH THEN
	LogEv(EL_AlarmStop,EO_TBV,1,1,'Over_Temperature_Alarm');
END_IF

fALARM_PM(IN:=ALARM_PM);
IF fALARM_PM.EVH THEN
	LogEv(EL_AlarmStop,EO_PMV,1,1,'Under_Pressure_Alarm');
END_IF
*)
(*
fALARM_ALARM_PM_PB_TB(IN:=ALARM_PM_PB_TB);
IF fALARM_ALARM_PM_PB_TB.EVH THEN
	LogEv(EL_AlarmStop,EO_PMV,1,1,'Allarmi_ISPESL');
END_IF
*)





(****************************************)

(*### VPN Connection Check ###*)
fVPN_ST1(IN:=VPN_ST1);
IF fVPN_ST1.EVH THEN
	LogEv(EL_Log,EO_VPN,1,1,'CONNECT_ON');
END_IF
IF fVPN_ST1.EVL THEN
	LogEv(EL_Log,EO_VPN,1,2,'CONNECT_OFF');
END_IF
(*
(*### VPN Status Check ###*)
fVPN_ST2(IN:=VPN_ST2);
IF fVPN_ST2.EVH THEN
	LogEv(EL_Log,EO_VPN,1,3,'STATUS_UP');
END_IF
IF fVPN_ST2.EVL THEN
	LogEv(EL_Wrn,EO_VPN,1,4,'STATUS_DOWN');
END_IF

(*### DOOR01 Status Check ###*)
fKEY_CT_ST(IN:=KEY_CT_ST);
IF fKEY_CT_ST.EVH THEN
	LogEv(EL_Log,EO_DOOR,1,2,'Centrale_termica_Close');
END_IF
IF fKEY_CT_ST.EVL THEN
	LogEv(EL_Wrn,EO_DOOR,1,1,'Centrale_termica_Open');
END_IF

(*### DOOR02 Status Check ###*)
fKEY_SCT_ST(IN:=KEY_SCT_ST);
IF fKEY_SCT_ST.EVH THEN
	LogEv(EL_Log,EO_DOOR,2,2,'Sottocentrale_termica_Close');
END_IF
IF fKEY_SCT_ST.EVL THEN
	LogEv(EL_Wrn,EO_DOOR,2,1,'Sottocentrale_termica_Open');
END_IF
*)
(*### DOOR03 Status Check ###*)
fKEY_QE_ST(IN:=KEY_QE_ST);
IF fKEY_QE_ST.EVH THEN
	LogEv(EL_Log,EO_DOOR,3,2,'Quadro_Close');
END_IF
IF fKEY_QE_ST.EVL THEN
	LogEv(EL_Wrn,EO_DOOR,3,1,'Quadro_Open');
END_IF
END_PROGRAM

(* POU Utils/USRLED_Update, ST *)
PROGRAM USRLED_Update
VAR
	OldStatus: en_SYS_Status;

	aFS : ARRAY [0..24] OF FLASHING_SEQUENCE :=
		(Colour:=GREEN,  Frequency:=1,   Relation:=128, Duration:=t#0s,    NextIndex:=0),  (* 0 => RUNNING *)
		(Colour:=ORANGE, Frequency:=1,   Relation:=128, Duration:=t#0s,    NextIndex:=1),  (* 1 => INIT *)
		(Colour:=RED,    Frequency:=4,   Relation:=128, Duration:=t#0s,    NextIndex:=2),  (* 2 => ERROR *)
		(Colour:=RED,    Frequency:=10,  Relation:=128, Duration:=t#0s,    NextIndex:=3),  (* 3 => ALARM *)
		(Colour:=ORANGE, Frequency:=200, Relation:=16,  Duration:=t#100ms, NextIndex:=11), (* 10 *)
		(Colour:=ORANGE, Frequency:=200, Relation:=32,  Duration:=t#100ms, NextIndex:=12),
		(Colour:=ORANGE, Frequency:=200, Relation:=64,  Duration:=t#100ms, NextIndex:=13),
		(Colour:=ORANGE, Frequency:=200, Relation:=128, Duration:=t#100ms, NextIndex:=14),
		(Colour:=ORANGE, Frequency:=200, Relation:=192, Duration:=t#100ms, NextIndex:=15),
		(Colour:=ORANGE, Frequency:=200, Relation:=128, Duration:=t#100ms, NextIndex:=16),
		(Colour:=ORANGE, Frequency:=200, Relation:=64,  Duration:=t#100ms, NextIndex:=17),
		(Colour:=ORANGE, Frequency:=200, Relation:=32,  Duration:=t#100ms, NextIndex:=18),
		(Colour:=ORANGE, Frequency:=200, Relation:=16,  Duration:=t#100ms, NextIndex:=19),
		(Colour:=ORANGE, Frequency:=200, Relation:=8,   Duration:=t#100ms, NextIndex:=10),
		(Colour:=GREEN,  Frequency:=200, Relation:=16,  Duration:=t#100ms, NextIndex:=21), (* 20 *)
		(Colour:=GREEN,  Frequency:=200, Relation:=32,  Duration:=t#100ms, NextIndex:=22),
		(Colour:=GREEN,  Frequency:=200, Relation:=64,  Duration:=t#100ms, NextIndex:=23),
		(Colour:=GREEN,  Frequency:=200, Relation:=128, Duration:=t#100ms, NextIndex:=24),
		(Colour:=GREEN,  Frequency:=200, Relation:=192, Duration:=t#100ms, NextIndex:=25),
		(Colour:=GREEN,  Frequency:=200, Relation:=128, Duration:=t#100ms, NextIndex:=26),
		(Colour:=GREEN,  Frequency:=200, Relation:=64,  Duration:=t#100ms, NextIndex:=27),
		(Colour:=GREEN,  Frequency:=200, Relation:=32,  Duration:=t#100ms, NextIndex:=28),
		(Colour:=GREEN,  Frequency:=200, Relation:=16,  Duration:=t#100ms, NextIndex:=29),
		(Colour:=GREEN,  Frequency:=200, Relation:=8,   Duration:=t#100ms, NextIndex:=20);

	pFS : POINTER TO FLASHING_SEQUENCE;


END_VAR
IF Sys.Status <> OldStatus THEN

	OldStatus:=Sys.Status;

	CASE OldStatus OF

		S_STARTUP:
			pFS:=ADR(aFS);
			SET_FLASHING_SEQUENCE(EN:=TRUE, POINTER_TO_POINTER_TO_ARRAY:=ADR(pFS));
			SET_FLASHING_SEQUENCE_INDEX(EN:=TRUE, IMMEDIATE:=FALSE, INDEX:=1);
			START_FLASHING_SEQUENCE(EN:=TRUE);

		S_RUNNING:
			SET_FLASHING_SEQUENCE_INDEX(EN:=TRUE, IMMEDIATE:=TRUE, INDEX:=0);

	END_CASE

END_IF
END_PROGRAM

(* POU ClevergyBlocks/OBJ_ANZ_INEPRO_PRO380/ANZ_INEPRO_DefineRegisters, ST *)
FUNCTION ANZ_INEPRO_DefineRegisters : BOOL
VAR_INPUT
END_VAR
VAR
	i:INT;
END_VAR
FOR I:=1 TO Plant_ANZ_inepro DO

MODBUS_INEPRO_RegAddress[i,1]:=16#2008;
MODBUS_INEPRO_RegDescr[i,1]:='L1 Voltage';
MODBUS_INEPRO_RegQuantity[i,1]:=2;
MODBUS_INEPRO_RegValueType[i,1]:=VALUE_REAL;

MODBUS_INEPRO_RegAddress[i,2]:=16#200C;
MODBUS_INEPRO_RegDescr[i,2]:='L2 Voltage';
MODBUS_INEPRO_RegQuantity[i,2]:=2;
MODBUS_INEPRO_RegValueType[i,2]:=VALUE_REAL;

MODBUS_INEPRO_RegAddress[i,3]:=16#2010;
MODBUS_INEPRO_RegDescr[i,3]:='L3 Voltage';
MODBUS_INEPRO_RegQuantity[i,3]:=2;
MODBUS_INEPRO_RegValueType[i,3]:=VALUE_REAL;

MODBUS_INEPRO_RegAddress[i,4]:=16#2020;
MODBUS_INEPRO_RegDescr[i,4]:='Grid frequency';
MODBUS_INEPRO_RegQuantity[i,4]:=2;
MODBUS_INEPRO_RegValueType[i,4]:=VALUE_REAL;

MODBUS_INEPRO_RegAddress[i,5]:=16#2068;
MODBUS_INEPRO_RegDescr[i,5]:='L1 CURRENT';
MODBUS_INEPRO_RegQuantity[i,5]:=2;
MODBUS_INEPRO_RegValueType[i,5]:=VALUE_REAL;

MODBUS_INEPRO_RegAddress[i,6]:=16#206C;
MODBUS_INEPRO_RegDescr[i,6]:='L2 CURRENT';
MODBUS_INEPRO_RegQuantity[i,6]:=2;
MODBUS_INEPRO_RegValueType[i,6]:=VALUE_REAL;

MODBUS_INEPRO_RegAddress[i,7]:=16#2070;
MODBUS_INEPRO_RegDescr[i,7]:='L3 CURRENT';
MODBUS_INEPRO_RegQuantity[i,7]:=2;
MODBUS_INEPRO_RegValueType[i,7]:=VALUE_REAL;

MODBUS_INEPRO_RegAddress[i,8]:=16#2080;
MODBUS_INEPRO_RegDescr[i,8]:='ACTIVE POWER';
MODBUS_INEPRO_RegQuantity[i,8]:=2;
MODBUS_INEPRO_RegValueType[i,8]:=VALUE_REAL;

MODBUS_INEPRO_RegAddress[i,9]:=16#2088;
MODBUS_INEPRO_RegDescr[i,9]:='L1 ACTIVE POWER';
MODBUS_INEPRO_RegQuantity[i,9]:=2;
MODBUS_INEPRO_RegValueType[i,9]:=VALUE_REAL;

MODBUS_INEPRO_RegAddress[i,10]:=16#208C;
MODBUS_INEPRO_RegDescr[i,10]:='L2 ACTIVE POWER';
MODBUS_INEPRO_RegQuantity[i,10]:=2;
MODBUS_INEPRO_RegValueType[i,10]:=VALUE_REAL;

MODBUS_INEPRO_RegAddress[i,11]:=16#2090;
MODBUS_INEPRO_RegDescr[i,11]:='L3 ACTIVE POWER';
MODBUS_INEPRO_RegQuantity[i,11]:=2;
MODBUS_INEPRO_RegValueType[i,11]:=VALUE_REAL;

MODBUS_INEPRO_RegAddress[i,12]:=16#20A0;
MODBUS_INEPRO_RegDescr[i,12]:='REACTIVE POWER';
MODBUS_INEPRO_RegQuantity[i,12]:=2;
MODBUS_INEPRO_RegValueType[i,12]:=VALUE_REAL;

MODBUS_INEPRO_RegAddress[i,13]:=16#20A8;
MODBUS_INEPRO_RegDescr[i,13]:='L1 REACTIVE POWER';
MODBUS_INEPRO_RegQuantity[i,13]:=2;
MODBUS_INEPRO_RegValueType[i,13]:=VALUE_REAL;

MODBUS_INEPRO_RegAddress[i,14]:=16#20AC;
MODBUS_INEPRO_RegDescr[i,14]:='L2 REACTIVE POWER';
MODBUS_INEPRO_RegQuantity[i,14]:=2;
MODBUS_INEPRO_RegValueType[i,14]:=VALUE_REAL;

MODBUS_INEPRO_RegAddress[i,15]:=16#20B0;
MODBUS_INEPRO_RegDescr[i,15]:='L3 REACTIVE POWER';
MODBUS_INEPRO_RegQuantity[i,15]:=2;
MODBUS_INEPRO_RegValueType[i,15]:=VALUE_REAL;

MODBUS_INEPRO_RegAddress[i,16]:=16#20C0;
MODBUS_INEPRO_RegDescr[i,16]:='APPARENT POWER';
MODBUS_INEPRO_RegQuantity[i,16]:=2;
MODBUS_INEPRO_RegValueType[i,16]:=VALUE_REAL;

MODBUS_INEPRO_RegAddress[i,17]:=16#20C8;
MODBUS_INEPRO_RegDescr[i,17]:='L1 APPARENT POWER';
MODBUS_INEPRO_RegQuantity[i,17]:=2;
MODBUS_INEPRO_RegValueType[i,17]:=VALUE_REAL;

MODBUS_INEPRO_RegAddress[i,18]:=16#20CC;
MODBUS_INEPRO_RegDescr[i,18]:='L2 APPARENT POWER';
MODBUS_INEPRO_RegQuantity[i,18]:=2;
MODBUS_INEPRO_RegValueType[i,18]:=VALUE_REAL;

MODBUS_INEPRO_RegAddress[i,19]:=16#20D0;
MODBUS_INEPRO_RegDescr[i,19]:='L3 APPARENT POWER';
MODBUS_INEPRO_RegQuantity[i,19]:=2;
MODBUS_INEPRO_RegValueType[i,19]:=VALUE_REAL;

MODBUS_INEPRO_RegAddress[i,20]:=16#20E0;
MODBUS_INEPRO_RegDescr[i,20]:='POWER FACTOR';
MODBUS_INEPRO_RegQuantity[i,20]:=2;
MODBUS_INEPRO_RegValueType[i,20]:=VALUE_REAL;

MODBUS_INEPRO_RegAddress[i,21]:=16#20E8;
MODBUS_INEPRO_RegDescr[i,21]:='L1 POWER FACTOR';
MODBUS_INEPRO_RegQuantity[i,21]:=2;
MODBUS_INEPRO_RegValueType[i,21]:=VALUE_REAL;

MODBUS_INEPRO_RegAddress[i,22]:=16#20EC;
MODBUS_INEPRO_RegDescr[i,22]:='L2 POWER FACTOR';
MODBUS_INEPRO_RegQuantity[i,22]:=2;
MODBUS_INEPRO_RegValueType[i,22]:=VALUE_REAL;

MODBUS_INEPRO_RegAddress[i,23]:=16#20F0;
MODBUS_INEPRO_RegDescr[i,23]:='L3 POWER FACTOR';
MODBUS_INEPRO_RegQuantity[i,23]:=2;
MODBUS_INEPRO_RegValueType[i,23]:=VALUE_REAL;

MODBUS_INEPRO_RegAddress[i,24]:=16#3000;
MODBUS_INEPRO_RegDescr[i,24]:='TOTAL ACTIVE ENERGY';
MODBUS_INEPRO_RegQuantity[i,24]:=2;
MODBUS_INEPRO_RegValueType[i,24]:=VALUE_REAL;

MODBUS_INEPRO_RegAddress[i,25]:=16#3060;
MODBUS_INEPRO_RegDescr[i,25]:='TOTAL REACTIVE ENERGY';
MODBUS_INEPRO_RegQuantity[i,25]:=2;
MODBUS_INEPRO_RegValueType[i,25]:=VALUE_REAL;

MODBUS_INEPRO_RegAddress[i,26]:=16#1000;
MODBUS_INEPRO_RegDescr[i,26]:='SERIAL_NUMBER';
MODBUS_INEPRO_RegQuantity[i,26]:=2;
MODBUS_INEPRO_RegValueType[i,26]:=VALUE_LONG;

END_FOR
END_FUNCTION

(* POU Utils Functions/AVERAGE_T, ST *)
FUNCTION_BLOCK AVERAGE_T
VAR_INPUT
	IN: 	INT;
END_VAR
VAR_OUTPUT
	HI:		INT;
	AVG:	INT;
	LOW:	INT;
	ERR:	BOOL;
END_VAR
VAR
	sum:	DINT;
	cnt:	WORD;
END_VAR
IF cnt>=65000 THEN
	ERR:=TRUE;
	Read();
	sum := sum - AVG;
	cnt := cnt + 1;
END_IF

sum := sum + IN;
cnt := cnt + 1;

IF IN<LOW THEN  LOW:=IN; END_IF
IF IN>HI  THEN HI :=IN; END_IF
END_FUNCTION_BLOCK
ACTION Read:
AVG := DINT_TO_INT(sum/cnt);
END_ACTION
ACTION Reset:
HI:=IN;
AVG:=IN;
LOW:=IN;
ERR:=FALSE;

sum:=IN;
cnt:=1;
END_ACTION

(* POU ClevergyBlocks/OBJ_ANZ_INEPRO_PRO380/BUILD_REAL_COPY, ST *)
FUNCTION BUILD_REAL_COPY : REAL
VAR_INPUT
		W1	:	WORD;
		W2	:	WORD;
END_VAR
VAR
 	awWords      : ARRAY[1..2] OF WORD;
  	pReal : POINTER TO REAL;
  	rReal : REAL;
END_VAR
awWords[1] := W1;
awWords[2] := W2;
pReal := ADR(awWords);
rReal := pReal^;
BUILD_REAL_COPY:=rReal;
END_FUNCTION

(* POU Utils Functions/COPY_32SWAP16, ST *)
FUNCTION COPY_32SWAP16:BOOL
VAR_INPUT
	pSourceAddress		:POINTER TO ARRAY[1..2] OF WORD;
	pDestinationAddress	:POINTER TO ARRAY[1..2] OF WORD;
END_VAR
VAR
END_VAR
pDestinationAddress^[1]:=pSourceAddress^[2];
pDestinationAddress^[2]:=pSourceAddress^[1];
END_FUNCTION

(* POU Utils Functions/FLT_EVENT, ST *)
FUNCTION_BLOCK FLT_EVENT
VAR_INPUT
	IN		: BOOL;
	INITEV	: BOOL:=TRUE;
END_VAR
VAR_OUTPUT
	EVH		: BOOL;
	EVL		: BOOL;
END_VAR
VAR
	init	: BOOL:=FALSE;
	old		: BOOL;
END_VAR
EVH:=FALSE;
EVL:=FALSE;

IF NOT init THEN
	init:=TRUE;
	IF INITEV THEN
		old := NOT IN;
	ELSE
		old := IN;
	END_IF
END_IF

IF old<>IN THEN
	old:=IN;
	IF IN THEN EVH:=TRUE; ELSE EVL:=TRUE; END_IF
END_IF
END_FUNCTION_BLOCK

(* POU Utils Functions/FLT_TIME, ST *)
FUNCTION_BLOCK FLT_TIME
VAR_INPUT
	IN		: BOOL;
	TTAP	: TIME:=T#5s;
	INITEV	: BOOL:=TRUE;
END_VAR
VAR_OUTPUT
	OUT		: BOOL;
	EVH		: BOOL;
	EVL		: BOOL;
END_VAR
VAR
	init	: BOOL:=FALSE;
	timer	: TON;
END_VAR
EVH:=FALSE;
EVL:=FALSE;

IF NOT init THEN
	init := TRUE;
	IF INITEV THEN
		OUT  := NOT IN;
	ELSE
		OUT  := IN;
	END_IF
END_IF

IF OUT<>IN THEN
	timer(IN:=TRUE,PT:=TTAP);
	IF timer.Q THEN
		OUT:=IN;
		timer(IN:=FALSE);
		IF OUT THEN EVH:=TRUE; ELSE EVL:=TRUE; END_IF
	END_IF
ELSE
	timer(IN:=FALSE);
END_IF
END_FUNCTION_BLOCK

(* POU Utils/FUN_ByteAsci, ST *)
FUNCTION FUN_ByteAsci : STRING(1)
VAR_INPUT
	ByteIn:BYTE;
END_VAR
VAR
END_VAR
CASE ByteIn OF

	32: FUN_ByteAsci:=' ';
	33: FUN_ByteAsci:='!';
	34: FUN_ByteAsci:='"';
	35: FUN_ByteAsci:='#';

	37: FUN_ByteAsci:='%';
	38: FUN_ByteAsci:='&';

	40: FUN_ByteAsci:='(';
	41: FUN_ByteAsci:=')';
	42: FUN_ByteAsci:='*';
	43: FUN_ByteAsci:='+';
	44: FUN_ByteAsci:=',';
	45: FUN_ByteAsci:='-';
	46: FUN_ByteAsci:='.';
	47: FUN_ByteAsci:='/';
	48: FUN_ByteAsci:='0';
	49: FUN_ByteAsci:='1';
	50: FUN_ByteAsci:='2';
	51: FUN_ByteAsci:='3';
	52: FUN_ByteAsci:='4';
	53: FUN_ByteAsci:='5';
	54: FUN_ByteAsci:='6';
	55: FUN_ByteAsci:='7';
	56: FUN_ByteAsci:='8';
	57: FUN_ByteAsci:='9';
	58: FUN_ByteAsci:=':';
	59: FUN_ByteAsci:=';';
	60: FUN_ByteAsci:='<';
	61: FUN_ByteAsci:='=';
	62: FUN_ByteAsci:='>';
	63: FUN_ByteAsci:='?';
	64: FUN_ByteAsci:='@';
	65: FUN_ByteAsci:='A';
	66: FUN_ByteAsci:='B';
	67: FUN_ByteAsci:='C';
	68: FUN_ByteAsci:='D';
	69: FUN_ByteAsci:='E';
	70: FUN_ByteAsci:='F';
	71: FUN_ByteAsci:='G';
	72: FUN_ByteAsci:='H';
	73: FUN_ByteAsci:='I';
	74: FUN_ByteAsci:='J';
	75: FUN_ByteAsci:='K';
	76: FUN_ByteAsci:='L';
	77: FUN_ByteAsci:='M';
	78: FUN_ByteAsci:='N';
	79: FUN_ByteAsci:='O';
	80: FUN_ByteAsci:='P';
	81: FUN_ByteAsci:='Q';
	82: FUN_ByteAsci:='R';
	83: FUN_ByteAsci:='S';
	84: FUN_ByteAsci:='T';
	85: FUN_ByteAsci:='U';
	86: FUN_ByteAsci:='V';
	87: FUN_ByteAsci:='W';
	88: FUN_ByteAsci:='X';
	89: FUN_ByteAsci:='Y';
	90: FUN_ByteAsci:='Z';
	91: FUN_ByteAsci:='[';
	92: FUN_ByteAsci:='\';
	93: FUN_ByteAsci:=']';
	94: FUN_ByteAsci:='^';
	95: FUN_ByteAsci:='_';
	96: FUN_ByteAsci:='`';
	97: FUN_ByteAsci:='a';
	98: FUN_ByteAsci:='b';
	99: FUN_ByteAsci:='c';
	100: FUN_ByteAsci:='d';
	101: FUN_ByteAsci:='e';
	102: FUN_ByteAsci:='f';
	103: FUN_ByteAsci:='g';
	104: FUN_ByteAsci:='h';
	105: FUN_ByteAsci:='i';
	106: FUN_ByteAsci:='j';
	107: FUN_ByteAsci:='k';
	108: FUN_ByteAsci:='l';
	109: FUN_ByteAsci:='m';
	110: FUN_ByteAsci:='n';
	111: FUN_ByteAsci:='o';
	112: FUN_ByteAsci:='p';
	113: FUN_ByteAsci:='q';
	114: FUN_ByteAsci:='r';
	115: FUN_ByteAsci:='s';
	116: FUN_ByteAsci:='t';
	117: FUN_ByteAsci:='u';
	118: FUN_ByteAsci:='v';
	119: FUN_ByteAsci:='w';
	120: FUN_ByteAsci:='x';
	121: FUN_ByteAsci:='y';
	122: FUN_ByteAsci:='z';
	123: FUN_ByteAsci:='{';
	124: FUN_ByteAsci:='|';
	125: FUN_ByteAsci:='}';
	126: FUN_ByteAsci:='~';

	167: FUN_ByteAsci:='°';
	176: FUN_ByteAsci:='°';


ELSE
	FUN_ByteAsci:='';

END_CASE
END_FUNCTION

(* POU Utils Functions/FUN_DEAD_ZONE, ST *)
FUNCTION FUN_DEAD_ZONE : INT
VAR_INPUT
	X : INT;
	L : INT;
END_VAR
VAR
	DEAD_BAND: BOOL;
END_VAR
IF X>=FUN_DEAD_ZONE+L THEN
	FUN_DEAD_ZONE := X ;
ELSIF X <= FUN_DEAD_ZONE-L THEN
	FUN_DEAD_ZONE := X;
ELSE
	FUN_DEAD_ZONE :=FUN_DEAD_ZONE;
END_IF;
END_FUNCTION

(* POU Utils Functions/LAMP_AL_GENERALE, ST *)
FUNCTION_BLOCK LAMP_AL_GENERALE
VAR_INPUT

	Allarme: BOOL;
	Warning: BOOL;
END_VAR
VAR_OUTPUT
	SistemaOK:BOOL;
	SistemaInAllarme:BOOL;
	SistemaWarning:BOOL;
	AllarmeLampada:BOOL;
END_VAR
VAR
	Lampeggio:BLINK;
END_VAR
IF Allarme THEN       					(* Se Allarme Attivo Lucde fissa ON *)
	SistemaInAllarme:=TRUE;
	SistemaWarning:=FALSE;
	AllarmeLampada:=TRUE;
ELSIF Warning THEN					(* Se Allarme Attivo Lucde fissa pulse *)
	SistemaInAllarme:=FALSE;
	SistemaWarning:=TRUE;
	Lampeggio(ENABLE:=TRUE , TIMELOW:=t#1s , TIMEHIGH:=t#1s , OUT=>AllarmeLampada );
ELSE
	SistemaInAllarme:=FALSE;
	SistemaWarning:=FALSE;
	AllarmeLampada:=FALSE;
END_IF
END_FUNCTION_BLOCK

(* POU Utils Functions/LINEAR_BAD, ST *)
FUNCTION LINEAR_BAD : INT (* Linear interpolation *)
VAR_INPUT
	PuntoMinX	: INT;
	PuntoMaxX	: INT;
	ValIn		: INT;
	PuntoMinY	: REAL;
	PuntoMaxY	: REAL;
	Decimali	: BYTE;
END_VAR
VAR
	Gain				: REAL;
	PuntoMinX_R			: REAL;
	PuntoMaxX_R			: REAL;
	Linearizzazione_R	: REAL;
END_VAR
PuntoMinX_R:=INT_TO_REAL(PuntoMinX);
PuntoMaxX_R:=INT_TO_REAL(PuntoMaxX);

Gain:=(PuntoMaxX_R-PuntoMinX_R)/(PuntoMaxY-PuntoMinY);	(* Calcolo in guadagno per la linarizzazione *)
Linearizzazione_R:=PuntoMinx+(Gain*(ValIn-PuntoMinY));	(* Ottengo il valore linearizzato *)

LINEAR_BAD:=REAL_TO_INT(Linearizzazione_R*(EXPT(10, Decimali)));  (* Ottengo intero con i decimai voluti *)
END_FUNCTION

(* POU Utils Functions/MEMCLR, ST *)
FUNCTION MEMCLR:BOOL
VAR_INPUT
	pDestinationAddress:POINTER TO ARRAY[1..2] OF BYTE;
	BytesToClear:WORD;
END_VAR
VAR
END_VAR
WHILE (BytesToClear > 0) DO
	pDestinationAddress^[1]:=0;
	pDestinationAddress:=ADR(pDestinationAddress^[2]); (* increment destination *)
	BytesToClear:=BytesToClear -1; (* decrement number of bytes to copy *)
END_WHILE
END_FUNCTION

(* POU Plant_Objects/obj_AI_GEN, ST *)
FUNCTION_BLOCK obj_AI_GEN
(* === TEMPERATURE PROBE FROM ANALOG INPUT ===
   v1.0[16/04/05] - Versioning
*)
VAR_INPUT
	(* Settings *)
	ID				: BYTE;
	PuntoMinX		: INT;			(* Parametri per la scalatura *)
	PuntoMaxX		: INT;
	PuntoMinY		: REAL;
	PuntoMaxY		: REAL;
	Decimali		: BYTE:=1;
	SogliaHH		: WORD;			(* Soglia per segnalazione Allarme Extra Range in alto - Solitamente sondo in CC *)
	SogliaHL		: WORD;			(* Soglia per segnalazione Allarme Extra Range in Basso - Solitamente sondo Aperta *)
	SogliaWH		: REAL;			(* Soglia per segnalazione Warning  in alto  *)
	SogliaWL		: REAL;    		(* Soglia per segnalazione Warning in basso  *)
	TAP				: INT:=2000;	(* Filtro in msec *)
	INITEV			: BOOL:= TRUE;	(* Generate init OK event *)
	(* Physical input *)
	AI_INPUT		: WORD;    		(* Sensor analog input *)
	TipoSensore:STRING(12);
END_VAR
VAR_OUTPUT
	WRN				: BOOL;	(* Segnalazione Warning *)
	ERR				: BOOL; (* Segnalazione Errore *)
	ValoreScalato	: INT;
	(* Status *)
	Status_Log	: BYTE;
	Status_Vis 	: DWORD;
END_VAR
VAR
	SegnaleHH	: BOOL;
	SegnaleHL	: BOOL;
	SegnaleOK	: BOOL;
	SegnaleWH	: BOOL;
	SegnaleWL	: BOOL;
    FiltroWRN	: TON;
    FiltroOK	: TON;
    FiltroERR	: TON;
END_VAR
(* Verifico che le variabile letta dall'ingresso Analogico  sia dentro i range
ATTENZIONE I LIMITI SPESSO SONO IN WORD VERIFICA  TABELLA MANUALE WAGO  *)

SegnaleHH:=(AI_INPUT>=SogliaHH);
SegnaleHL:=(AI_INPUT<=SogliaHL);
SegnaleOK:=NOT (SegnaleHH OR SegnaleHL);

(* Linerarizzo il segnale di ingresso e la converto in unita ingegneristiche *)
ValoreScalato:=LINEAR_BAD(PuntoMinX, PuntoMaxX, AI_INPUT, PuntoMinY, PuntoMaxY, Decimali);


IF SegnaleOK  THEN
	(*  Verifica  e segnalazione Warning *)
	SegnaleWH:=(ValoreScalato>SogliaWH*(EXPT(10, Decimali)));
	SegnaleWL:=(ValoreScalato<SogliaWL*(EXPT(10, Decimali)));

	Status_Log:=0;
	Status_Vis:=16#20F020;    (* Indicazione WEB Visu Sonda OK *)

	FiltroWRN( IN:=(SegnaleWH OR SegnaleWL), PT:=INT_TO_TIME(TAP) );    (* Filtro su LOG *)
	IF  FiltroWRN.Q THEN     (* Condizione di WARNING *)
		IF NOT WRN THEN
			WRN:=TRUE;
			Status_Log:=1;
			LogEv(EL_Wrn,EO_TPV,ID,SEL(ValoreScalato<=SogliaWL,3,2),INT_TO_STRING(ValoreScalato));
		END_IF
	END_IF

    IF (INITEV OR WRN OR ERR) AND NOT FiltroWRN.Q THEN
		FiltroWRN(IN:=FALSE  , PT:=INT_TO_TIME(TAP));    (* Resetto il Filtro su LOG WRN  *)
		FiltroERR(IN:=FALSE  , PT:=INT_TO_TIME(TAP));    (* Resetto il Filtro su LOG ERR *)
		INITEV:=FALSE; ERR:=FALSE; WRN:=FALSE;
		LogEv(EL_Log,EO_TPV,ID,1,'');
	END_IF
ELSE
	FiltroERR(IN:=TRUE  , PT:= INT_TO_TIME(TAP) );    (* Filtro su LOG *)
	IF  FiltroERR.Q THEN     (* Condizione di WARNING *)
		IF NOT ERR THEN
			ERR:=TRUE;
			Status_Log:=2;

			IF SegnaleHH THEN LogEv(EL_Alarm,EO_TPV,ID,6,INT_TO_STRING(ValoreScalato));END_IF;
			IF SegnaleHL THEN LogEv(EL_Alarm,EO_TPV,ID,4,INT_TO_STRING(ValoreScalato));END_IF;
		END_IF
	END_IF

	Status_Vis:=16#2020F0;   (* Indicazione WEB Visu Sonda KO *)
END_IF



(* Status Log *)
IF ERR THEN
	Status_Log := 2;
	Status_Vis := COLOR_RED;
ELSIF WRN THEN
	Status_Log := 1;
	Status_Vis := COLOR_YELLOW;
ELSE
	Status_Log := 0; Status_Vis := COLOR_GREEN;
END_IF
END_FUNCTION_BLOCK
ACTION AddLogData:
Logger.s1:=CONCAT('&',TipoSensore);
IF ID<10 THEN Logger.s1:=CONCAT(Logger.s1,'0');END_IF
Logger.s1:=CONCAT(Logger.s1,BYTE_TO_STRING(ID));
Logger.s1:=CONCAT(Logger.s1,'=');


Logger.s1:=CONCAT(Logger.s1,WORD_TO_STRING(Status_Log));		Logger.s1:=CONCAT(Logger.s1,';');
Logger.s1:=CONCAT(Logger.s1,INT_TO_STRING(ValoreScalato));


ADDSTRING(ADR(Logger.TData), ADR(Logger.s1), Logger.TLen);
END_ACTION

(* POU ClevergyBlocks/OBJ_ANZ_INEPRO_PRO380/obj_ANZ_INEPRO_PRO380, ST *)
FUNCTION_BLOCK obj_ANZ_INEPRO_PRO380
(* === Block for realizing the ANZ entity with the meter INEPRO PRO380 ===
	
	One ANZ block manages one physical ANZ device.
	
	Versioning:
		v1.0 [28/07/16] - Diego Bernini
*)
VAR_INPUT

	(* Logical ID of the ANZ, univocal w.r.t the plant *)
	ID										 : WORD;
	(* Type of ANZ: 1-phase or 3-phase *)
	contabilizerMode							 : en_ANZ_Type := THREE_PHASE;

	modbusConnector: obj_MODBUS_GENERIC_CONNECTOR;

	(* meter dependent fields, by the connector*)
	specificData								:  typ_ANZ_INEPRO_PRO380;

	(* determines if warning errors are sent or not *)
	enableWarning : BOOL :=FALSE;

	TIMING_AGGREGATED_MEASURE:TIME;
	TIMING_RESET_AGGREGATED_MEASURE:TIME;

END_VAR

VAR_OUTPUT

	(* output records representing the data in according to the ANZ Clevergy Web format *)
	measures						: typ_ANZ_real;
	(*status of the block according the Clevergy architecture *)
	Status_Log						: BYTE;
	Status_Vis	:	DWORD;

END_VAR

VAR

	contAvg								 : REAL :=0;
	sumAvg								 : REAL :=0;
	timerCalc								 : TON;
	timerReset							 : TON;

	alarmMsg : STRING;
	alarmLaunched: ARRAY[1..MAX_ALARM] OF BYTE;

	warningMsg : STRING;
	warningLaunched: ARRAY[1..MAX_WARNING] OF BYTE;

	i : BYTE;
	tmpAlarm:BYTE;
	tmpWarning:BYTE;

END_VAR
VAR CONSTANT
	MAX_ALARM :BYTE:=20;
	MAX_WARNING :BYTE:=20;
END_VAR
VAR
	CheckEvents: BOOL;
END_VAR
Status_Log:=ModBusConnector.Status_Log;

getModbusData();

timerReset(IN:=NOT timerReset.Q,PT:=TIMING_RESET_AGGREGATED_MEASURE);
IF timerReset.Q THEN

	sumAvg := 0;
	contAvg := 0;

 	specificData.rMaximumTotalActivePower:=0; (* reset => min possible val *)
	specificData.rMaximumTotalReactivePower:= -2147483648;
	specificData.rMaximumCurrentL1:=0;
	specificData.rMaximumCurrentL2:=0;
	specificData.rMaximumCurrentL3:=0;

END_IF

(*compute additional measures, the ones which are not provided directly*)
timerCalc(IN:=NOT timerCalc.Q,PT:=TIMING_AGGREGATED_MEASURE);

IF timerCalc.Q THEN
	sumAvg := sumAvg+specificData.rTotalActivePower;
	contAvg:=contAvg+1;
	specificData.rAverageTotalActivePower:=sumAvg/contAvg;
	IF specificData.rTotalActivePower > specificData.rMaximumTotalActivePower THEN specificData.rMaximumTotalActivePower:= specificData.rTotalActivePower; END_IF
	IF specificData.rTotalReactivePower > specificData.rMaximumTotalReactivePower THEN specificData.rMaximumTotalReactivePower:= specificData.rTotalReactivePower; END_IF

	IF specificData.arCurrent[1] > specificData.rMaximumCurrentL1 THEN specificData.rMaximumCurrentL1:= specificData.arCurrent[1]; END_IF
	IF specificData.arCurrent[2] > specificData.rMaximumCurrentL2 THEN specificData.rMaximumCurrentL2:= specificData.arCurrent[2]; END_IF
	IF specificData.arCurrent[3] > specificData.rMaximumCurrentL3 THEN specificData.rMaximumCurrentL3:= specificData.arCurrent[3]; END_IF

END_IF


(* convert the data to the Clevergy format *)
convertToClevergyFormat();

(* visu	*)
IF Status_Log = 2 THEN
	Status_Vis := COLOR_RED;
ELSIF Status_Log = 1 THEN
	Status_Vis := COLOR_YELLOW;
ELSE
	Status_Vis := COLOR_GREEN;
END_IF
END_FUNCTION_BLOCK
ACTION AddLogData:
Logger.s1:=INSERT('&ANZ=',WORD_TO_STRING(ID),4);
IF ID<10 THEN Logger.s1:=INSERT(Logger.s1,'0',4); END_IF

Logger.s1:=CONCAT(Logger.s1,REAL_TO_STRING(measures.V_L1N));		Logger.s1:=CONCAT(Logger.s1,';');
Logger.s1:=CONCAT(Logger.s1,REAL_TO_STRING(measures.V_L2N));		Logger.s1:=CONCAT(Logger.s1,';');
Logger.s1:=CONCAT(Logger.s1,REAL_TO_STRING(measures.V_L3N));		Logger.s1:=CONCAT(Logger.s1,';');
Logger.s1:=CONCAT(Logger.s1,REAL_TO_STRING(measures.V_L1L2));		Logger.s1:=CONCAT(Logger.s1,';');
Logger.s1:=CONCAT(Logger.s1,REAL_TO_STRING(measures.V_L2L3));		Logger.s1:=CONCAT(Logger.s1,';');
Logger.s1:=CONCAT(Logger.s1,REAL_TO_STRING(measures.V_L3L1));		Logger.s1:=CONCAT(Logger.s1,';');

Logger.s1:=CONCAT(Logger.s1,REAL_TO_STRING(measures.FREQ));		Logger.s1:=CONCAT(Logger.s1,';');

Logger.s1:=CONCAT(Logger.s1,REAL_TO_STRING(measures.I_L1));		Logger.s1:=CONCAT(Logger.s1,';');
Logger.s1:=CONCAT(Logger.s1,REAL_TO_STRING(measures.I_L2));		Logger.s1:=CONCAT(Logger.s1,';');
Logger.s1:=CONCAT(Logger.s1,REAL_TO_STRING(measures.I_L3));		Logger.s1:=CONCAT(Logger.s1,';');
Logger.s1:=CONCAT(Logger.s1,REAL_TO_STRING(measures.I_L1_Max)); 	Logger.s1:=CONCAT(Logger.s1,';');
Logger.s1:=CONCAT(Logger.s1,REAL_TO_STRING(measures.I_L2_Max)); 	Logger.s1:=CONCAT(Logger.s1,';');
Logger.s1:=CONCAT(Logger.s1,REAL_TO_STRING(measures.I_L3_Max)); 	Logger.s1:=CONCAT(Logger.s1,';');

Logger.s1:=CONCAT(Logger.s1,REAL_TO_STRING(measures.PF_L1));		Logger.s1:=CONCAT(Logger.s1,';');
Logger.s1:=CONCAT(Logger.s1,REAL_TO_STRING(measures.PF_L2));		Logger.s1:=CONCAT(Logger.s1,';');
Logger.s1:=CONCAT(Logger.s1,REAL_TO_STRING(measures.PF_L3));		Logger.s1:=CONCAT(Logger.s1,';');

Logger.s1:=CONCAT(Logger.s1,REAL_TO_STRING(measures.P_3P));		Logger.s1:=CONCAT(Logger.s1,';');
Logger.s1:=CONCAT(Logger.s1,REAL_TO_STRING(measures.P_3P_Avg)); 	Logger.s1:=CONCAT(Logger.s1,';');
Logger.s1:=CONCAT(Logger.s1,REAL_TO_STRING(measures.P_3P_Max)); 	Logger.s1:=CONCAT(Logger.s1,';');

Logger.s1:=CONCAT(Logger.s1,REAL_TO_STRING(measures.Q_3P));			Logger.s1:=CONCAT(Logger.s1,';');
Logger.s1:=CONCAT(Logger.s1, REAL_TO_STRING(measures.Q_3P_Max));		Logger.s1:=CONCAT(Logger.s1,';');

Logger.s1:=CONCAT(Logger.s1,REAL_TO_STRING(measures.WH_3P));			Logger.s1:=CONCAT(Logger.s1,';');
Logger.s1:=CONCAT(Logger.s1,REAL_TO_STRING(measures.VARH_3P));			Logger.s1:=CONCAT(Logger.s1,';');

Logger.s1:=CONCAT(Logger.s1,BYTE_TO_STRING(Status_Log)); 					Logger.s1:=CONCAT(Logger.s1,';');

Logger.s1:=CONCAT(Logger.s1,REAL_TO_STRING(measures.COSPHI_L1));		Logger.s1:=CONCAT(Logger.s1,';');
Logger.s1:=CONCAT(Logger.s1,REAL_TO_STRING(measures.COSPHI_L2));		Logger.s1:=CONCAT(Logger.s1,';');
Logger.s1:=CONCAT(Logger.s1,REAL_TO_STRING(measures.COSPHI_L3));		Logger.s1:=CONCAT(Logger.s1,';');

Logger.s1:=CONCAT(Logger.s1,BYTE_TO_STRING(SEL(contabilizerMode=THREE_PHASE,1,0)));

ADDSTRING(ADR(Logger.TData), ADR(Logger.s1), Logger.TLen);
END_ACTION
ACTION AddLogData_OLD:
(*Logger.s1:=INSERT('&ANZ=',WORD_TO_STRING(ID),4);
IF ID<10 THEN Logger.s1:=INSERT(Logger.s1,'0',4); END_IF

Logger.s1:=CONCAT(Logger.s1,DWORD_TO_STRING(measures.V_L1N));		Logger.s1:=CONCAT(Logger.s1,';');
Logger.s1:=CONCAT(Logger.s1,DWORD_TO_STRING(measures.V_L2N));		Logger.s1:=CONCAT(Logger.s1,';');
Logger.s1:=CONCAT(Logger.s1,DWORD_TO_STRING(measures.V_L3N));		Logger.s1:=CONCAT(Logger.s1,';');
Logger.s1:=CONCAT(Logger.s1,DWORD_TO_STRING(measures.V_L1L2));		Logger.s1:=CONCAT(Logger.s1,';');
Logger.s1:=CONCAT(Logger.s1,DWORD_TO_STRING(measures.V_L2L3));		Logger.s1:=CONCAT(Logger.s1,';');
Logger.s1:=CONCAT(Logger.s1,DWORD_TO_STRING(measures.V_L3L1));		Logger.s1:=CONCAT(Logger.s1,';');

Logger.s1:=CONCAT(Logger.s1,DWORD_TO_STRING(measures.FREQ));		Logger.s1:=CONCAT(Logger.s1,';');

Logger.s1:=CONCAT(Logger.s1,DWORD_TO_STRING(measures.I_L1));		Logger.s1:=CONCAT(Logger.s1,';');
Logger.s1:=CONCAT(Logger.s1,DWORD_TO_STRING(measures.I_L2));		Logger.s1:=CONCAT(Logger.s1,';');
Logger.s1:=CONCAT(Logger.s1,DWORD_TO_STRING(measures.I_L3));		Logger.s1:=CONCAT(Logger.s1,';');
Logger.s1:=CONCAT(Logger.s1,DWORD_TO_STRING(measures.I_L1_Max)); 	Logger.s1:=CONCAT(Logger.s1,';');
Logger.s1:=CONCAT(Logger.s1,DWORD_TO_STRING(measures.I_L2_Max)); 	Logger.s1:=CONCAT(Logger.s1,';');
Logger.s1:=CONCAT(Logger.s1,DWORD_TO_STRING(measures.I_L3_Max)); 	Logger.s1:=CONCAT(Logger.s1,';');

Logger.s1:=CONCAT(Logger.s1,DINT_TO_STRING(measures.PF_L1));		Logger.s1:=CONCAT(Logger.s1,';');
Logger.s1:=CONCAT(Logger.s1,DINT_TO_STRING(measures.PF_L2));		Logger.s1:=CONCAT(Logger.s1,';');
Logger.s1:=CONCAT(Logger.s1,DINT_TO_STRING(measures.PF_L3));		Logger.s1:=CONCAT(Logger.s1,';');

Logger.s1:=CONCAT(Logger.s1,DINT_TO_STRING(measures.P_3P));		Logger.s1:=CONCAT(Logger.s1,';');
Logger.s1:=CONCAT(Logger.s1,DINT_TO_STRING(measures.P_3P_Avg)); 	Logger.s1:=CONCAT(Logger.s1,';');
Logger.s1:=CONCAT(Logger.s1,DINT_TO_STRING(measures.P_3P_Max)); 	Logger.s1:=CONCAT(Logger.s1,';');

Logger.s1:=CONCAT(Logger.s1,DINT_TO_STRING(measures.Q_3P));			Logger.s1:=CONCAT(Logger.s1,';');
Logger.s1:=CONCAT(Logger.s1,DINT_TO_STRING(measures.Q_3P_Max));		Logger.s1:=CONCAT(Logger.s1,';');

Logger.s1:=CONCAT(Logger.s1,DWORD_TO_STRING(measures.WH_3P));			Logger.s1:=CONCAT(Logger.s1,';');
Logger.s1:=CONCAT(Logger.s1,DINT_TO_STRING(measures.VARH_3P));			Logger.s1:=CONCAT(Logger.s1,';');

Logger.s1:=CONCAT(Logger.s1,BYTE_TO_STRING(Status_Log)); 					Logger.s1:=CONCAT(Logger.s1,';');

Logger.s1:=CONCAT(Logger.s1,DINT_TO_STRING(measures.COSPHI_L1));		Logger.s1:=CONCAT(Logger.s1,';');
Logger.s1:=CONCAT(Logger.s1,DINT_TO_STRING(measures.COSPHI_L2));		Logger.s1:=CONCAT(Logger.s1,';');
Logger.s1:=CONCAT(Logger.s1,DINT_TO_STRING(measures.COSPHI_L3));		Logger.s1:=CONCAT(Logger.s1,';');

Logger.s1:=CONCAT(Logger.s1,BYTE_TO_STRING(SEL(contabilizerMode=THREE_PHASE,1,0)));

ADDSTRING(ADR(Logger.TData), ADR(Logger.s1), Logger.TLen);*)
;
END_ACTION
ACTION checkAlarm:
(*IF(alarmLaunched[1]=0 AND typ_750_494_State.xPhase1_OverCurrentSystem) THEN
	alarmLaunched[1]:=2;
	LogEv(EL_Alarm,EO_ANZ,ID,3, 'xPhase1_OverCurrentSystem');
ELSIF (alarmLaunched[1]=2 AND NOT(typ_750_494_State.xPhase1_OverCurrentSystem) ) THEN
	alarmLaunched[1]:=0;
	LogEv(EL_Log,EO_ANZ,ID,4,'xPhase1_OverCurrentSystem');
END_IF*)

;
END_ACTION
ACTION checkEventsToSignal:
CheckAlarm();
CheckWarning();
CheckStatus();
END_ACTION
ACTION checkStatus:
(*tmpAlarm:=0;
FOR I:=1 TO MAX_alarm DO tmpAlarm:=tmpAlarm+alarmLaunched[i]; END_FOR
IF(tmpAlarm>0) THEN status_Log:=2; END_IF

tmpWarning:=0;
FOR I:=1 TO MAX_WARNING DO tmpWarning:=tmpWarning+warningLaunched[i]; END_FOR
IF(status=0 AND tmpWarning>0) THEN status:=1; END_IF

IF (tmpAlarm =0 AND tmpWarning =0) THEN status:=0; END_IF*)
;
END_ACTION
ACTION checkWarning:
IF(enableWarning = FALSE) THEN RETURN; END_IF

(*IF( warningLaunched[1]=0 AND typ_750_494_State.xGeneralError) THEN
	warningLaunched[1]:=2;
	LogEv(EL_Wrn,EO_ANZ,ID,5, 'xGeneralError');
ELSIF (warningLaunched[1]=2 AND NOT(typ_750_494_State.xGeneralError) ) THEN
	warningLaunched[1]:=0;
	LogEv(EL_Log,EO_ANZ,ID,5,'xGeneralError');
END_IF*)

;
END_ACTION
ACTION convertToClevergyFormat:
	measures.V_L1N := specificData.arVoltage_L_N[1];
	measures.V_L2N := specificData.arVoltage_L_N[2];
	measures.V_L3N := specificData.arVoltage_L_N[3];

	(*n/a*)
	measures.V_L1L2:=0;
	measures.V_L2L3:=0;
	measures.V_L3L1:=0;

	measures.FREQ := specificData.arFrequency*1000;

	measures.I_L1 := specificData.arCurrent[1]*1000;
	measures.I_L2 := specificData.arCurrent[2]*1000;
	measures.I_L3 :=specificData.arCurrent[3]*1000;

	measures.I_L1_Max := specificData.rMaximumCurrentL1*1000;
	measures.I_L2_Max := specificData.rMaximumCurrentL2*1000;
	measures.I_L3_Max := specificData.rMaximumCurrentL3*1000;

	measures.PF_L1 := specificData.arPowerFactorPF[1]*1000;
	measures.PF_L2 := specificData.arPowerFactorPF[2]*1000;
	measures.PF_L3 := specificData.arPowerFactorPF[3]*1000;

	measures.P_3P := specificData.rTotalActivePower*1000;
	measures.P_3P_Avg:=specificData.rAverageTotalActivePower*1000;
	measures.P_3P_Max:=specificData.rMaximumTotalActivePower*1000;

	measures.Q_3P:=specificData.rTotalReactivePower*1000;
	measures.Q_3P_Max:=specificData.rMaximumTotalReactivePower*1000;

	measures.WH_3P:=specificData.rTotalActiveEnergy*10;
	measures.VARH_3P:=specificData.rTotalReactiveEnergy*10;

	(*n/a*)
	measures.COSPHI_L1:=0;
	measures.COSPHI_L2:=0;
	measures.COSPHI_L3:=0;
END_ACTION
ACTION convertToClevergyFormat_OLD:
	measures.V_L1N := REAL_TO_DWORD(specificData.arVoltage_L_N[1]);
	measures.V_L2N := REAL_TO_DWORD(specificData.arVoltage_L_N[2]);
	measures.V_L3N := REAL_TO_DWORD(specificData.arVoltage_L_N[3]);

	(*n/a*)
	measures.V_L1L2:=REAL_TO_DWORD(0);
	measures.V_L2L3:=REAL_TO_DWORD(0);
	measures.V_L3L1:=REAL_TO_DWORD(0);

	measures.FREQ := REAL_TO_DWORD(specificData.arFrequency*1000);

	measures.I_L1 := REAL_TO_DWORD(specificData.arCurrent[1]*1000);
	measures.I_L2 := REAL_TO_DWORD(specificData.arCurrent[2]*1000);
	measures.I_L3 := REAL_TO_DWORD(specificData.arCurrent[3]*1000);

	measures.I_L1_Max := REAL_TO_DWORD(specificData.rMaximumCurrentL1*1000);
	measures.I_L2_Max := REAL_TO_DWORD(specificData.rMaximumCurrentL2*1000);
	measures.I_L3_Max := REAL_TO_DWORD(specificData.rMaximumCurrentL3*1000);

	measures.PF_L1 := REAL_TO_DINT(specificData.arPowerFactorPF[1]*1000);
	measures.PF_L2 := REAL_TO_DINT(specificData.arPowerFactorPF[2]*1000);
	measures.PF_L3 := REAL_TO_DINT(specificData.arPowerFactorPF[3]*1000);

	measures.P_3P := REAL_TO_DINT(specificData.rTotalActivePower);
	measures.P_3P_Avg:=REAL_TO_DINT(specificData.rAverageTotalActivePower);
	measures.P_3P_Max:=REAL_TO_DINT(specificData.rMaximumTotalActivePower);

	measures.Q_3P:=REAL_TO_DINT(specificData.rTotalReactivePower);
	measures.Q_3P_Max:=REAL_TO_DINT(specificData.rMaximumTotalReactivePower);

	measures.WH_3P:=REAL_TO_DINT(specificData.rTotalActiveEnergy*10);
	measures.VARH_3P:=REAL_TO_DINT(specificData.rTotalReactiveEnergy*10);

	(*n/a*)
	measures.COSPHI_L1:=REAL_TO_DINT(0);
	measures.COSPHI_L2:=REAL_TO_DINT(0);
	measures.COSPHI_L3:=REAL_TO_DINT(0);
;
END_ACTION
ACTION getModbusData:
specificData.arFrequency:=modBusConnector.regData[4];

specificData.arVoltage_L_N[1]:=modBusConnector.regData[1];
specificData.arVoltage_L_N[2]:=modBusConnector.regData[2];
specificData.arVoltage_L_N[3]:=modBusConnector.regData[3];

specificData.arCurrent[1]:=modBusConnector.regData[5];
specificData.arCurrent[2]:=modBusConnector.regData[6];
specificData.arCurrent[3]:=modBusConnector.regData[7];

specificData.rTotalActivePower:=modBusConnector.regData[8];
specificData.arActivePower[1]:=modBusConnector.regData[9];
specificData.arActivePower[2]:=modBusConnector.regData[10];
specificData.arActivePower[3]:=modBusConnector.regData[11];

specificData.rTotalReactivePower:=modBusConnector.regData[12];
specificData.arReactivePower[1]:=modBusConnector.regData[13];
specificData.arReactivePower[2]:=modBusConnector.regData[14];
specificData.arReactivePower[3]:=modBusConnector.regData[15];

specificData.rTotalApparentPower:=modBusConnector.regData[16];
specificData.arApparentPower[1]:=modBusConnector.regData[17];
specificData.arApparentPower[2]:=modBusConnector.regData[18];
specificData.arApparentPower[3]:=modBusConnector.regData[19];

specificData.rTotalPowerFactorPF:=modBusConnector.regData[20];
specificData.arPowerFactorPF[1]:=modBusConnector.regData[21];
specificData.arPowerFactorPF[2]:=modBusConnector.regData[22];
specificData.arPowerFactorPF[3]:=modBusConnector.regData[23];

specificData.rTotalActiveEnergy:=modBusConnector.regData[24];

specificData.rTotalReactiveEnergy:=modBusConnector.regData[25];
END_ACTION

(* POU ClevergyBlocks/OBJ_ANZ_INEPRO_PRO380/obj_MODBUS_GENERIC_CONNECTOR, ST *)
FUNCTION_BLOCK obj_MODBUS_GENERIC_CONNECTOR
VAR CONSTANT
		(* States of normal modbus data reading *)
		WAIT_STATE			:	BYTE := 0;
		QUERY_START_CYCLE	: 	BYTE := 1;
		QUERY_MEAS_REQ		:  	BYTE := 2;
		QUERY_MEAS_ANSW	: 	BYTE := 3;
		ERROR_STATE			:	BYTE := 4;
END_VAR
VAR_INPUT
		PARENT_EO_TYPE 		: 	WORD;
		PARENT_EO_ID		:	BYTE;
		Address				:	BYTE;
		TIMING				:	TIME:=t#500ms;

		retryErrMax			:	BYTE := 10;

END_VAR
VAR_IN_OUT
		ModBus		:	obj_MODBUS_ANZ;
END_VAR
VAR_OUTPUT
		Status_Log	:	BYTE;
		Status_Vis	:	DWORD;

		regDescr : ARRAY[1..MODBUS_INEPRO_MAX_REG] OF STRING(20);
		regAddress : ARRAY[1..MODBUS_INEPRO_MAX_REG] OF WORD;
		regQuantity : ARRAY[1..MODBUS_INEPRO_MAX_REG] OF BYTE;
		regValueType : ARRAY[1..MODBUS_INEPRO_MAX_REG] OF en_Modbus_Reg_Type;
		regData: ARRAY[1..MODBUS_INEPRO_MAX_REG] OF REAL;
		regDataWord: ARRAY[1..MODBUS_INEPRO_MAX_REG, 1..2] OF WORD;

END_VAR
VAR
		InitOK		:	BOOL := FALSE;

		(* Modbus State machine variables	*)
		state		:	BYTE;
		last_state		:	BYTE;
		retry		:	BYTE;
		retryErr		:	BYTE;
		ReadTmr		:	TON := (PT:=t#5s);	(* Just to do a first ModBus read at the beginning *)
		fModbusAlr	:	BOOL;

		(* Event check variable	*)
		Alarm		:	FLT_EVENT;
		ModBusAlr	:	FLT_EVENT := (INITEV:=FALSE);
		StatusOK		:	FLT_EVENT := (INITEV:=FALSE);
		AlarmCtr		:	BYTE;
		WarningCtr	:	BYTE;

		fTimeout	:	BOOL;

		currentReg:INT:=1;

		i:INT;
		x:INT;
END_VAR
IF NOT InitOK THEN
	ReadTmr.PT := timing;
	InitOK := TRUE;
	initMapping();
END_IF

(* State machine *)
Stm();

(* Check if an alarm has occured *)
CheckAlarm();

(* Set "Status_Log" according to actual object status	*)
IF AlarmCtr > 0 THEN
	Status_Log := 2;
	Status_Vis := COLOR_RED;
ELSIF WarningCtr > 0 THEN
	Status_Log := 1;
	Status_Vis := COLOR_YELLOW;
ELSE
	Status_Log := 0;

	Status_Vis := COLOR_GREEN;
END_IF
END_FUNCTION_BLOCK
ACTION CheckAlarm:
(*** Verify ModBus error	***)
ModbusAlr(IN:=fModbusAlr);

IF ModbusAlr.EVH THEN
	LogEv(EL_Alarm,PARENT_EO_TYPE,PARENT_EO_ID,2,SEL(ModBus.MB_MASTER.MB_Error<>0,'0','1'));
	AlarmCtr := AlarmCtr + 1;
END_IF

IF ModbusAlr.EVL THEN
	LogEv(EL_Log,PARENT_EO_TYPE,PARENT_EO_ID,1,'');
	AlarmCtr := SEL(AlarmCtr=0, AlarmCtr-1, 0);
END_IF
END_ACTION
ACTION initMapping:
FOR I:=1 TO MODBUS_INEPRO_MAX_REG DO

	IF MODBUS_INEPRO_RegAddress[PARENT_EO_ID,i] <> 0 THEN

		regAddress[i]:=MODBUS_INEPRO_RegAddress[PARENT_EO_ID, i];
		REGDescr[i]:=MODBUS_INEPRO_REGDescr[PARENT_EO_ID, i];
		regQuantity[i]:=MODBUS_INEPRO_regQuantity[PARENT_EO_ID, i];
		regValueType[i]:=MODBUS_INEPRO_regValueType[PARENT_EO_ID, i];

	END_IF

END_FOR
END_ACTION
ACTION Stm:
CASE state OF

	WAIT_STATE:	(* Refresh time manager *)

		ReadTmr(IN:=NOT(ReadTmr.Q));
		IF ReadTmr.Q THEN

			ReadTmr.PT := timing;			(* Refresh timer range *)

			(* Reset state machine variables and counters *)
			retry	:= 0;
			last_state	:= WAIT_STATE;

			(* Start state machine	*)
			state := QUERY_START_CYCLE;

		END_IF

	QUERY_START_CYCLE:
		IF NOT ModBus.MB_Start AND (NOT ModBus.MB_Lock OR retry>0) THEN
			ModBus.MB_Lock := TRUE;

			ModBus.MB_Obj := PARENT_EO_TYPE;
			ModBus.MB_ObjId := PARENT_EO_ID;

			state := QUERY_MEAS_REQ;
		END_IF

	(****			 MEASUREMENTS			  ****)

	QUERY_MEAS_REQ:
		IF NOT ModBus.MB_Start THEN

				IF regAddress[currentReg] <> 0 THEN

					ModBus.MB_Query.SlaveAddress := Address;
					ModBus.MB_Query.FunctionCode := 16#3;
					ModBus.MB_Query.Read_StartAddress :=regAddress[currentReg];
					ModBus.MB_Query.Read_Quantity := regQuantity[currentReg];
					ModBus.MB_Start := TRUE;

					state := QUERY_MEAS_ANSW;

				ELSE

					currentReg:=currentReg+1;

					IF(currentReg<=MODBUS_INEPRO_MAX_REG) THEN

						state := QUERY_MEAS_REQ;

					ELSE

						currentReg:=1;
						fModbusAlr := FALSE;
						retryErr := 0;
						ModBus.MB_Lock := FALSE;
						fTimeout := FALSE;
						state := WAIT_STATE;

					END_IF

				END_IF
		END_IF


	QUERY_MEAS_ANSW:
		IF NOT ModBus.MB_Start THEN
			IF ModBus.MB_MASTER.bInterfaceError<>0 OR ModBus.MB_MASTER.MB_Error<>0 THEN
				last_state := QUERY_MEAS_ANSW;
				state := ERROR_STATE;
			ELSE

				IF (regValueType[currentReg] = VALUE_REAL ) THEN
					regData[currentReg]:=BUILD_REAL_COPY(ModBus.MB_Resp.Data[1],ModBus.MB_Resp.Data[0]);
				END_IF
				IF (regValueType[currentReg] = VALUE_LONG ) THEN
					regDataWord[currentReg,1]:=ModBus.MB_Resp.Data[0];
					regDataWord[currentReg,2]:=ModBus.MB_Resp.Data[1];
				END_IF

				currentReg:=currentReg+1;

				IF(currentReg<=MODBUS_INEPRO_MAX_REG) THEN

					state := QUERY_MEAS_REQ;

				ELSE
					currentReg:=1;
					fModbusAlr := FALSE;
					retryErr := 0;
					ModBus.MB_Lock := FALSE;
					fTimeout := FALSE;
					state := WAIT_STATE;
				END_IF


			END_IF
		END_IF


	ERROR_STATE:	(* Error state *)

		IF retry < 3 THEN
			retry := retry+1;
			state := last_state;

		ELSE
			ModBus.MB_Lock := FALSE;

			(* Verify if slave is dead *)
			IF retryErr < retryErrMaX THEN
				retryErr := retryErr + 1;
			ELSE
				fModbusAlr := TRUE;
			END_IF

			(* Back to wait state *)
			state := WAIT_STATE;

			fTimeout := TRUE;
		END_IF

		IF ModBus.MB_MASTER.MB_Error=MB_TIME_OUT THEN
			state := state;
		END_IF
ELSE
	state := WAIT_STATE;
END_CASE
END_ACTION

(* POU ClevergyBlocks/obj_MODBUS_ANZ, ST *)
FUNCTION_BLOCK obj_MODBUS_ANZ
(* === MODBUS PROTOCOL INTERFACE ===
   v1.1[19/06/15] - Added new VARS allocation and searching
*)
VAR CONSTANT
	VARS_Max	: BYTE := 32;
END_VAR
VAR_INPUT
	(* Settings *)
	ID			: BYTE;
	COM			: BYTE;
	BAUDRATE	: COM_BAUDRATE;
	RS485		: BOOL := FALSE;
	PARITY : COM_PARITY:=PARITY_NO;
	STOP_BITS :COM_STOPBITS:=STOPBITS_2;
	TIME_OUT_TIME : TIME:=t#500ms;

	(* Interface *)
	MB_MASTER	: MODBUS_EXTENDED_MASTER;
	MB_Start	: BOOL;
	MB_Query	: typModbusExtendedQuery;
	MB_Resp		: typModbusResponse;
	MB_Lock		: BOOL;
	MB_Obj		: en_SYS_Objects;
	MB_ObjId	: BYTE;

	(* Variables management *)
	VARS_En		: BOOL := FALSE;
	VARS		: ARRAY [0..VARS_Max] OF typ_MODBUS_VAR_anz;
	VARS_Check	: BOOL;
	VARS_Alarm	: BOOL;

	(* Variables allocation *)
	VAR_Pointer : POINTER TO ARRAY[0..99] OF WORD;
	VAR_Cfg		: POINTER TO typ_MODBUS_VAR_ANZ;
END_VAR
VAR_OUTPUT
	(* Status *)
	Status_Log	: BYTE;
	Status_Vis	: DWORD;
END_VAR
VAR
	sta         : BYTE :=0;
	i			: BYTE;
	j			: BYTE;

	AlarmCOM	: FLT_EVENT;	(* Physical error relative to serial port -> COM	*)
	AlarmMDB	: FLT_EVENT;	(* ModBus error due to communication protocol error	*)

	VarTmr		: TON := (PT:=T#1s);
	VarSta		: BYTE; (* Status *)
	VarCnt		: BYTE; (* Scan counter *)
	VarRetry	: BYTE;
	VarAlarm	: BYTE; (* Last variable with errors *)
END_VAR
MB_MASTER(ENABLE:=TRUE,	ASCII_Mode:=FALSE, bCOM_PORT:=COM, cbCOM_BAUDRATE:=BAUDRATE, cpCOM_PARITY:=PARITY,
		csCOM_STOPBITS:=STOP_BITS,	cbsCOM_BYTESIZE:=BS_8, cfCOM_FLOW_CONTROL:=SEL(RS485,NO_FLOW_CONTROL,HALFDUPLEX),
		tTIME_OUT:=TIME_OUT_TIME,	StartFunction:=MB_Start, ExtQuery:=MB_Query, Response:=MB_Resp);

(* Process variable management *)
IF VARS_En THEN VARS_Process(); END_IF

(* Check status *)
AlarmCOM(IN:=(MB_MASTER.bInterfaceError<>0));
IF AlarmCOM.EVH THEN
	LogEv(SEL(MB_MASTER.bInterfaceError<>3,EL_Wrn,EL_Alarm),EO_MODBUS,ID,1,BYTE_TO_STRING(MB_MASTER.bInterfaceError));
END_IF
IF AlarmCOM.EVL THEN								(* Trigger a fall edge: MODBUS back working *)
	LogEv(EL_Log,EO_MODBUS,ID,2,'MODBUS_OK');
END_IF

(* If VARS not active check if a protocol error has occured (if VARS active this check is already done in "VARS_Process"	*)
IF NOT VARS_En THEN

	AlarmMDB(IN:=(MB_MASTER.MB_Error<>0));
(*	IF AlarmMDB.EVH THEN
		LogEv(EL_Wrn,EO_MODBUS,ID,2,INT_TO_STRING(MB_MASTER.MB_Error));
	END_IF
	IF AlarmMDB.EVL THEN								(* Trigger a fall edge: MODBUS back working *)
		LogEv(EL_Log,EO_MODBUS,ID,2,'MODBUS_OK');
	END_IF
*)
END_IF

(* Log/visu status *)
IF AlarmCOM.IN THEN Status_Log:=2; Status_Vis:=COLOR_RED;
ELSIF Vars_Alarm OR AlarmMDB.IN THEN Status_Log:=1; Status_Vis:=COLOR_YELLOW;
ELSE Status_Log:=0; Status_Vis:=COLOR_GREEN;
END_IF
END_FUNCTION_BLOCK
ACTION VAR_Search:
(* Search VAR with specific pointer if not found return first free VAR
	[Last VAR is not active... used as safe area...] 
*)
j:=VARS_Max;
FOR i := 0 TO VARS_Max-1 DO
	IF VARS[i].Variable=0 AND j>i THEN j:=i; END_IF
	IF VARS[i].Variable=VAR_Pointer THEN
		VAR_Cfg:=ADR(VARS[i]);
		RETURN;
	END_IF
END_FOR
VAR_Cfg:=ADR(VARS[j]);
END_ACTION
ACTION VARS_Process:
(* Update var timers *)
VarTmr(IN:=(NOT VarTmr.Q));
IF VarTmr.Q THEN
	FOR i := 0 TO VARS_Max DO
		IF VARS[i].Refresh_Cnt>0 THEN VARS[i].Refresh_Cnt:=VARS[i].Refresh_Cnt-1; END_IF
	END_FOR
	VARS_Check:=TRUE;
END_IF


(* Process status *)
CASE VarSta OF
	0: (* === Init *)
		VarCnt:=0;
		VarSta:=1;

	1: (* === Wait check signal *)
		IF VARS_Check THEN				(* Decremented "Refresh_Cnt" *)
			VARS_Check:=FALSE;
			VarCnt:=0;
			VarSta:=2;
		END_IF

	2: (* === Check loop *)
		IF NOT (MB_Lock OR MB_Start) THEN
			WHILE VarCnt<=(VARS_Max-1) AND VarSta=2 DO
				(* Check only active vars *)
				IF VARS[VarCnt].Variable<>0 THEN			(* "Variable" is a pointer to word, so if 0 no address *)
					(* Check var auto-refresh on timer checks *)
					IF VARS[VarCnt].Refresh_Time>0 AND VARS[VarCnt].Refresh_Cnt=0 THEN
						VARS[VarCnt].Refresh_Cnt:=VARS[VarCnt].Refresh_Time;
						VarSta:=3;
					END_IF
					(* Check refresh for change or request *)
					CASE VARS[VarCnt].FunCode OF
						5,6,15,16: (* Write functions *)
							IF VARS[VarCnt].Variable_Size=1 THEN
								IF VARS[VarCnt].Variable^[0]<>VARS[VarCnt].Variable_Mirror THEN
									VARS[VarCnt].Variable_Mirror:=VARS[VarCnt].Variable^[0];
									VarSta:=3;
								END_IF
							ELSE
								IF VARS[VarCnt].Variable_Mirror<>0 THEN
									VARS[VarCnt].Variable_Mirror:=0;
									VarSta:=3;
								END_IF
							END_IF
						1,2,3,4: (* Read functions *)
							IF VARS[VarCnt].Variable_Mirror<>0 THEN
								VARS[VarCnt].Variable_Mirror:=0;
								VarSta:=3;
							END_IF
					END_CASE
				END_IF
				(* Process query *)
				IF VarSta=3 THEN
					MB_Lock:=TRUE;
					MB_Query.SlaveAddress:=VARS[VarCnt].SlaveAddress;
					MB_Query.FunctionCode:=VARS[VarCnt].FunCode;
					CASE VARS[VarCnt].FunCode OF
						16#5,16#6,16#F,16#10:
							MB_Query.Read_Quantity:=0;
							MB_Query.Read_StartAddress:=0;
							MB_Query.Write_StartAddress:=VARS[VarCnt].FunAddress;
							MB_Query.Write_Quantity:=VARS[VarCnt].Variable_Size;
							IF VARS[VarCnt].Variable_Size=200 THEN
								COPY_32SWAP16(VARS[VarCnt].Variable, ADR(MB_Query.Write_Data[0]));
							ELSIF VARS[VarCnt].Variable_Size>1 THEN
								MEMCPY(VARS[VarCnt].Variable, ADR(MB_Query.Write_Data[0]), 2*VARS[VarCnt].Variable_Size);
							ELSE
								MB_Query.Write_Data[0]:=VARS[VarCnt].Variable^[0];
							END_IF
						16#1,16#2,16#3,16#4:
							MB_Query.Read_StartAddress:=VARS[VarCnt].FunAddress;
							IF VARS[VarCnt].Variable_Size=200 THEN MB_Query.Read_Quantity:=2; ELSE
							  MB_Query.Read_Quantity:=VARS[VarCnt].Variable_Size;
							END_IF
							MB_Query.Write_StartAddress:=0;
							MB_Query.Write_Quantity:=0;
					END_CASE
					VarRetry:=0;
					MB_Start:=TRUE;
				ELSE
					VarCnt:=VarCnt+1;
				END_IF
			END_WHILE
			(* Check loop completed -> no actions *)
			IF VarSta=2 THEN VarSta:=1; END_IF
		END_IF

	3: (* === Wait & process MB response *)
		IF NOT MB_Start THEN
			IF MB_MASTER.MB_Error=0 THEN
				CASE VARS[VarCnt].FunCode OF
					1,2,3,4:
						IF VARS[VarCnt].Variable_Size=200 THEN
							COPY_32SWAP16(ADR(MB_Resp.Data), VARS[VarCnt].Variable);
						ELSIF VARS[VarCnt].Variable_Size>1 THEN
							MEMCPY(ADR(MB_Resp.Data), VARS[VarCnt].Variable, 2*VARS[VarCnt].Variable_Size);
						ELSE
							VARS[VarCnt].Variable^[0]:=MB_Resp.Data[0];
						END_IF
				END_CASE
				MB_Lock:=FALSE;
				(* Signal error recovery *)
				IF VARS_Alarm=TRUE AND VarCnt=VarAlarm THEN
					LogEv(EL_Wrn,EO_MODBUS,ID,5,'');
					VARS_Alarm:=FALSE;
				END_IF
				(* Next var *)
				VarCnt:=VarCnt+1;
				VarSta:=2;
			ELSE
				IF VarRetry<3 THEN
					VarRetry:=VarRetry+1;
					MB_Start:=TRUE;
				ELSE
					MB_Lock:=FALSE;
					(* Signal error *)
					IF VARS_Alarm=FALSE THEN
						LogEv(EL_Wrn,EO_MODBUS,ID,3,INT_TO_STRING(MB_MASTER.MB_Error));
						VARS_Alarm:=TRUE;
						VarAlarm:=VarCnt-1;
					END_IF
					(* Next var *)
					VarCnt:=VarCnt+1;
					VarSta:=2;
				END_IF
			END_IF
		END_IF

ELSE
	VarSta:=0;
END_CASE
END_ACTION

(* POU Plant_Objects/obj_COMPRESSORE_NEW, ST *)
FUNCTION_BLOCK obj_COMPRESSORE_NEW
VAR CONSTANT

	TimeOutModBus: TON;


END_VAR
VAR_INPUT
	ID			:	BYTE;
	Address		:	BYTE;


	(* Modbus *)
	Refresh_Now	:	BOOL;			(* Richiesta di lettura stato macchina Immediata  *)
	retryErrMax	:	BYTE := 2;

	OnOff		: 	BOOL;

	IndirizzoDaScrivere: WORD;
	DatoDaScrivere: INT;
	ScriviDato: BOOL;
	ScriviCoil: BOOL;

	fWriteAttivazioneComandi:BOOL;

	RUN_REQ: BOOL;
	STOP_REQ:BOOL;
	AgggiornoStartStop: BOOL;
	CARICO_REQ: BOOL;
	RELEASE_REQ: BOOL;


	LocSelManAuto:BOOL;
	LocTGP:INT;
	LocASP:INT;




END_VAR
VAR_IN_OUT
	ModBus		:obj_MODBUS;
END_VAR
VAR_OUTPUT
	Run			:	BOOL;

	Status_Log	:	WORD;
	Status_Vis	:	DWORD;
END_VAR
VAR
	(* da diego per gestione stato stringa > 255*)
	temp :STRING(255);
	tempRaw		: ARRAY [0..MAX_SEND_TCP_CLIENT] OF BYTE;
	tempRawLen :DINT;
	longString:STRING(255);

	(* Timer manage switch on/off delay *)
	Delay		: 	TONOF;
	Warning		:	FLT_TAP := (TAP:=100);
	AllarmeCompressore_MB		:	FLT_TAP;
	WarningCompressore_MB		:	FLT_TAP;
	AllarmeCompressoreAttivo_MB		:	FLT_TAP;
	RientrAllarmeCompressore_MB		:	FLT_TAP;
	RientrWarningCompressore_MB		:	FLT_TAP;
	AllarmeAttivo: INT;


	state		:	INT;
	retry		:	BYTE;
	retryErr	:	BYTE;
	ReadTmr		:	TON := (PT:=T#5s);
	fModbusAlr:BOOL;

	Ctrl_Run: BOOL;


	VerificaFuctionCode: INT;
	VerificaNodoLetto: INT;
	ErroreComuModBus: BOOL;
	IndiceErrore: BYTE;

	MB_BitStato: ARRAY [0..1] OF BOOL;
	MB_RegistriLetti: ARRAY [0..1] OF INT;
	MB_RegistriHoldingLetti: ARRAY [0..260] OF INT;
	MB_BitStatoCoil: ARRAY [0..1] OF BOOL;



	AddressRead: BYTE;
	index: BYTE;
	indexErr: BYTE;





	x: INT;

	IndirizzoStart: INT;
	Stop: BOOL;
	start: BOOL;
	StatusControl: ARRAY [0..15] OF BOOL;
	CompressoreInAllarme: BOOL;
	CompressoreInWarning: BOOL;

	AllarmeAttivoSuCompressore: INT;
	WarningAttivoSuCompressore: INT;
	TOFF_RitardoAllarme: TOF;
	TOFF_RitardoWarning: TOF;
END_VAR
(* Call ModBus state machine *)
Stm();

(* Check alarm	*)
CheckAlarm();

(* Seganalzione stato Compressore  *)
IF ErroreComuModBus OR AllarmeCompressoreAttivo_MB.IN THEN (* corretto da DB 27/07/2017, era AllarmeCompressore_MB*)
		Status_Log:=2; Status_Vis:=16#2020F0;
  ELSIF WarningCompressore_MB.IN  THEN
		Status_Log:=1; Status_Vis:=16#20F0F0;
    ELSE
		Status_Log:=0;
		Status_Vis:=16#006000;
END_IF
END_FUNCTION_BLOCK
ACTION AddLogData:
Logger.s1:=INSERT('&COMPINGRR=',BYTE_TO_STRING(ID),10);
IF ID<10 THEN Logger.s1:=INSERT(Logger.s1,'0',10); END_IF

FOR tempRawLen:=0 TO MAX_SEND_TCP_CLIENT DO
                tempRaw[tempRawLen]:=0;
END_FOR

tempRawLen:=0;


temp:=Logger.s1;
ADDSTRING(ADR(tempRaw), ADR(temp), tempRawLen);

temp:=CONCAT(WORD_TO_STRING(Status_Log),';');
ADDSTRING(ADR(tempRaw), ADR(temp), tempRawLen);


(* Sparo gli ingressi Digitali **)
FOR x:= 0 TO 15 DO
	temp:=CONCAT(SEL(StatusControl[x],'0','1'),';');
	ADDSTRING(ADR(tempRaw), ADR(temp), tempRawLen);
END_FOR

(*

temp:=CONCAT(INT_TO_STRING(MB_RegistriHoldingLetti[1]),';');
ADDSTRING(ADR(tempRaw), ADR(temp), tempRawLen); *)
temp:=CONCAT(INT_TO_STRING(MB_RegistriHoldingLetti[3]),';');
ADDSTRING(ADR(tempRaw), ADR(temp), tempRawLen);
temp:=CONCAT(INT_TO_STRING(MB_RegistriHoldingLetti[4]),';');
ADDSTRING(ADR(tempRaw), ADR(temp), tempRawLen);
temp:=CONCAT(INT_TO_STRING(MB_RegistriHoldingLetti[5]),';');
ADDSTRING(ADR(tempRaw), ADR(temp), tempRawLen);
temp:=CONCAT(INT_TO_STRING(MB_RegistriHoldingLetti[6]),';');
ADDSTRING(ADR(tempRaw), ADR(temp), tempRawLen);
temp:=CONCAT(INT_TO_STRING(MB_RegistriHoldingLetti[11]),';');
ADDSTRING(ADR(tempRaw), ADR(temp), tempRawLen);
temp:=CONCAT(INT_TO_STRING(MB_RegistriHoldingLetti[12]),';');
ADDSTRING(ADR(tempRaw), ADR(temp), tempRawLen);
temp:=CONCAT(INT_TO_STRING(MB_RegistriHoldingLetti[13]),';');
ADDSTRING(ADR(tempRaw), ADR(temp), tempRawLen);
temp:=CONCAT(INT_TO_STRING(MB_RegistriHoldingLetti[14]),';');
ADDSTRING(ADR(tempRaw), ADR(temp), tempRawLen);
temp:=CONCAT(INT_TO_STRING(MB_RegistriHoldingLetti[15]),';');
ADDSTRING(ADR(tempRaw), ADR(temp), tempRawLen);
temp:=CONCAT(INT_TO_STRING(MB_RegistriHoldingLetti[19]),';');
ADDSTRING(ADR(tempRaw), ADR(temp), tempRawLen);
temp:=CONCAT(INT_TO_STRING(MB_RegistriHoldingLetti[20]),';');
ADDSTRING(ADR(tempRaw), ADR(temp), tempRawLen);
temp:=CONCAT(INT_TO_STRING(MB_RegistriHoldingLetti[25]),';');
ADDSTRING(ADR(tempRaw), ADR(temp), tempRawLen);
temp:=CONCAT(INT_TO_STRING(MB_RegistriHoldingLetti[26]),';');
ADDSTRING(ADR(tempRaw), ADR(temp), tempRawLen);
temp:=CONCAT(INT_TO_STRING(MB_RegistriHoldingLetti[27]),';');
ADDSTRING(ADR(tempRaw), ADR(temp), tempRawLen);
temp:=CONCAT(INT_TO_STRING(MB_RegistriHoldingLetti[30]),';');
ADDSTRING(ADR(tempRaw), ADR(temp), tempRawLen);
temp:=CONCAT(INT_TO_STRING(MB_RegistriHoldingLetti[31]),';');
ADDSTRING(ADR(tempRaw), ADR(temp), tempRawLen);
temp:=CONCAT(INT_TO_STRING(MB_RegistriHoldingLetti[64]),';');
ADDSTRING(ADR(tempRaw), ADR(temp), tempRawLen);
temp:=CONCAT(INT_TO_STRING(MB_RegistriHoldingLetti[65]),';');
ADDSTRING(ADR(tempRaw), ADR(temp), tempRawLen);
temp:=CONCAT(INT_TO_STRING(MB_RegistriHoldingLetti[101]),';');
ADDSTRING(ADR(tempRaw), ADR(temp), tempRawLen);
temp:=CONCAT(INT_TO_STRING(MB_RegistriHoldingLetti[112]),';');
ADDSTRING(ADR(tempRaw), ADR(temp), tempRawLen);
temp:=CONCAT(INT_TO_STRING(MB_RegistriHoldingLetti[113]),';');
ADDSTRING(ADR(tempRaw), ADR(temp), tempRawLen);
temp:=CONCAT(INT_TO_STRING(MB_RegistriHoldingLetti[114]),';');
ADDSTRING(ADR(tempRaw), ADR(temp), tempRawLen);
temp:=CONCAT(INT_TO_STRING(MB_RegistriHoldingLetti[115]),';');
ADDSTRING(ADR(tempRaw), ADR(temp), tempRawLen);
temp:=CONCAT(INT_TO_STRING(MB_RegistriHoldingLetti[118]),';');
ADDSTRING(ADR(tempRaw), ADR(temp), tempRawLen);
temp:=CONCAT(INT_TO_STRING(MB_RegistriHoldingLetti[119]),';');
ADDSTRING(ADR(tempRaw), ADR(temp), tempRawLen);
temp:=CONCAT(INT_TO_STRING(MB_RegistriHoldingLetti[121]),';');
ADDSTRING(ADR(tempRaw), ADR(temp), tempRawLen);
temp:=CONCAT(INT_TO_STRING(MB_RegistriHoldingLetti[255]),';');
ADDSTRING(ADR(tempRaw), ADR(temp), tempRawLen);
temp:=(INT_TO_STRING(MB_RegistriHoldingLetti[256]));
ADDSTRING(ADR(tempRaw), ADR(temp), tempRawLen);


ADDSTRING(ADR(Logger.TData), ADR(tempRaw), Logger.TLen);
END_ACTION
ACTION CheckAlarm:
(**** GEstione Log ad Evento *****)




(*	AllarmeCompressore_MB(IN:=MB_RegistriHoldingLetti[1].6 );
	AllarmeCompressoreAttivo_MB(IN:=MB_RegistriHoldingLetti[1].6 AND MB_RegistriHoldingLetti[256]<>AllarmeAttivo ); *)

	AllarmeCompressoreAttivo_MB(IN:=CompressoreInAllarme AND AllarmeAttivoSuCompressore<>AllarmeAttivo );

	IF AllarmeCompressore_MB.EVH OR AllarmeCompressoreAttivo_MB.EVH THEN
		LogEv(EL_Alarm,EO_COMPINGRR,ID,1,CONCAT ('AllarmeAttivo_n.', INT_TO_STRING(MB_RegistriHoldingLetti[255])));
		AllarmeAttivo:=MB_RegistriHoldingLetti[256];
	END_IF

	TOFF_RitardoAllarme(in:=CompressoreInAllarme,pt:=t#10s);    (* AllarmeAttivoSuCompressore=0 *)
	RientrAllarmeCompressore_MB(IN:=(TOFF_RitardoAllarme.Q) );

	IF RientrAllarmeCompressore_MB.EVL THEN
		LogEv(EL_Log,EO_COMPINGRR,ID,2,CONCAT ('AllarmeRientrato_n.', INT_TO_STRING(MB_RegistriHoldingLetti[255])));
		AllarmeAttivo:=0;
		AllarmeAttivoSuCompressore:=0;
	END_IF



	WarningCompressore_MB(IN:=CompressoreInWarning );

	IF WarningCompressore_MB.EVH THEN
		LogEv(EL_Wrn,EO_COMPINGRR,ID,1,CONCAT ('AllarmeAttivo_n.', INT_TO_STRING(MB_RegistriHoldingLetti[255])));
	END_IF
	TOFF_RitardoWarning(in:=CompressoreInWarning,pt:=t#10s);   (* WarningAttivoSuCompressore=0*)
	RientrWarningCompressore_MB(IN:=(TOFF_RitardoWarning.Q) );

	IF RientrWarningCompressore_MB.EVL THEN
		LogEv(EL_Log,EO_COMPINGRR,ID,2,CONCAT ('AllarmeRientrato_n.', INT_TO_STRING(MB_RegistriHoldingLetti[255])));
	END_IF
END_ACTION
ACTION Stm:
CASE state OF
	0:	(* Refresh time manager *)
		ReadTmr(IN:=NOT ReadTmr.Q);
		(*A tempo interrogo il nodo sempre che non ci sia qualcuno che lo sta interrogando in quel momento *)

		IF (ReadTmr.Q AND NodoDaInterrogareCompressoreNuovo=Address )  AND NOT InibiscoModbusCompressoreNuovo THEN
			state := 10;
			ReadTmr.PT := T#100ms;  (* moreno *)
			Refresh_Now := FALSE;
			InibiscoModbusCompressoreNuovo := TRUE;
		END_IF

	(**** Leggo le Analogiche a Disposzione  ****)

	10:	(* richiedo lettura Holding Registere   *)

		Modbus.MB_Query.SlaveAddress := Address;
		Modbus.MB_Query.FunctionCode := 3;
		IndirizzoStart:=1;
		ModBus.MB_Query.Read_StartAddress :=IndirizzoStart - 1 ;
		ModBus.MB_Query.Read_Quantity := 19;(*19;*)
		ModBus.MB_Start := TRUE;
		state := 20;

	20:	(* Risposta all'interrogazione *)
		IF NOT ModBus.MB_Start   THEN
			VerificaFuctionCode:=ModBus.MB_Resp.FunctionCode;
			VerificaNodoLetto:=ModBus.MB_Resp.SlaveAddress;

			IF ModBus.MB_MASTER.MB_Error<>0 THEN
				state := 300;
			ELSE
				FOR x:=0 TO ModBus.MB_Query.Read_Quantity DO
					MB_RegistriHoldingLetti[x+IndirizzoStart] := ModBus.MB_Resp.Data[x];   	(* Vedi tabella *)
				END_FOR

				(* trasforo la wordo in singoli 16 bit *)

					StatusControl[0]:= MB_RegistriHoldingLetti[IndirizzoStart].0;   	(* Vedi tabella *)
					StatusControl[1]:= MB_RegistriHoldingLetti[IndirizzoStart].1;   	(* Vedi tabella *)
					StatusControl[2]:= MB_RegistriHoldingLetti[IndirizzoStart].2;   	(* Vedi tabella *)
					StatusControl[3]:= MB_RegistriHoldingLetti[IndirizzoStart].3;   	(* Vedi tabella *)
					StatusControl[4]:= MB_RegistriHoldingLetti[IndirizzoStart].4;   	(* Vedi tabella *)
					StatusControl[5]:= MB_RegistriHoldingLetti[IndirizzoStart].5;   	(* Vedi tabella *)
					StatusControl[6]:= MB_RegistriHoldingLetti[IndirizzoStart].6;   	(* Vedi tabella *)
					StatusControl[7]:= MB_RegistriHoldingLetti[IndirizzoStart].7;   	(* Vedi tabella *)
					StatusControl[8]:= MB_RegistriHoldingLetti[IndirizzoStart].8;   	(* Vedi tabella *)
					StatusControl[9]:= MB_RegistriHoldingLetti[IndirizzoStart].9;   	(* Vedi tabella *)
					StatusControl[10]:= MB_RegistriHoldingLetti[IndirizzoStart].10;   	(* Vedi tabella *)
					StatusControl[11]:= MB_RegistriHoldingLetti[IndirizzoStart].11;   	(* Vedi tabella *)
					StatusControl[12]:= MB_RegistriHoldingLetti[IndirizzoStart].12;   	(* Vedi tabella *)
					StatusControl[13]:= MB_RegistriHoldingLetti[IndirizzoStart].13;   	(* Vedi tabella *)
					StatusControl[14]:= MB_RegistriHoldingLetti[IndirizzoStart].14;   	(* Vedi tabella *)
					StatusControl[15]:= MB_RegistriHoldingLetti[IndirizzoStart].15;   	(* Vedi tabella *)

					CompressoreInAllarme:=StatusControl[6];
					CompressoreInWarning:=StatusControl[7];


				IndirizzoStart:=20;
				ModBus.MB_Query.Read_StartAddress :=IndirizzoStart - 1 ;
				ModBus.MB_Query.Read_Quantity := 19;
				ModBus.MB_Start := TRUE;

				state := 30;
			END_IF
		END_IF

	30: (* Rispota Altri paramenti *)
		IF NOT ModBus.MB_Start  THEN

			IF ModBus.MB_MASTER.MB_Error<>0 THEN
				state := 300;
			ELSE

				FOR x:=0 TO ModBus.MB_Query.Read_Quantity DO
					MB_RegistriHoldingLetti[x+IndirizzoStart] := ModBus.MB_Resp.Data[x];   	(* Vedi tabella *)
				END_FOR

				IndirizzoStart:=40;
				ModBus.MB_Query.Read_StartAddress :=IndirizzoStart - 1 ;
				ModBus.MB_Query.Read_Quantity := 19;
				ModBus.MB_Start := TRUE;

				state := 35;
			END_IF
		END_IF
	35: (* Rispota Altri paramenti *)
		IF NOT ModBus.MB_Start  THEN

			IF ModBus.MB_MASTER.MB_Error<>0 THEN
				state := 300;
			ELSE

				FOR x:=0 TO ModBus.MB_Query.Read_Quantity DO
					MB_RegistriHoldingLetti[x+IndirizzoStart] := ModBus.MB_Resp.Data[x];   	(* Vedi tabella *)
				END_FOR

				IndirizzoStart:=64;
				ModBus.MB_Query.Read_StartAddress :=IndirizzoStart - 1 ;
				ModBus.MB_Query.Read_Quantity := 6;
				ModBus.MB_Start := TRUE;

				state := 40;
			END_IF
		END_IF
	40: (* Rispota Altri paramenti *)
		IF NOT ModBus.MB_Start  THEN

			IF ModBus.MB_MASTER.MB_Error<>0 THEN
				state := 300;
			ELSE

				FOR x:=0 TO ModBus.MB_Query.Read_Quantity DO
					MB_RegistriHoldingLetti[x+IndirizzoStart] := ModBus.MB_Resp.Data[x];   	(* Vedi tabella *)
				END_FOR

				IndirizzoStart:=90;
				ModBus.MB_Query.Read_StartAddress :=IndirizzoStart - 1 ;
				ModBus.MB_Start := TRUE;

				state := 45;
			END_IF
		END_IF

	45: (* Rispota Altri paramenti *)
		IF NOT ModBus.MB_Start  THEN

			IF ModBus.MB_MASTER.MB_Error<>0 THEN
				state := 300;
			ELSE
				FOR x:=0 TO ModBus.MB_Query.Read_Quantity DO
					MB_RegistriHoldingLetti[x+IndirizzoStart] := ModBus.MB_Resp.Data[x];   	(* Vedi tabella *)
				END_FOR

				IndirizzoStart:=110;
				ModBus.MB_Query.Read_StartAddress :=IndirizzoStart - 1 ;
				ModBus.MB_Query.Read_Quantity := 19;
				ModBus.MB_Start := TRUE;

				state := 50;
			END_IF
		END_IF


	50: (* Rispota Altri paramenti *)
		IF NOT ModBus.MB_Start  THEN

			IF ModBus.MB_MASTER.MB_Error<>0 THEN
				state := 300;
			ELSE
				FOR x:=0 TO ModBus.MB_Query.Read_Quantity DO
					MB_RegistriHoldingLetti[x+IndirizzoStart] := ModBus.MB_Resp.Data[x];   	(* Vedi tabella *)
				END_FOR

				IndirizzoStart:=130;
				ModBus.MB_Query.Read_StartAddress :=IndirizzoStart - 1 ;
				ModBus.MB_Query.Read_Quantity := 5;
				ModBus.MB_Start := TRUE;


				state := 55;
			END_IF
		END_IF

	55: (* Rispota Altri paramenti *)
		IF NOT ModBus.MB_Start  THEN

			IF ModBus.MB_MASTER.MB_Error<>0 THEN
				state := 300;
			ELSE
				FOR x:=0 TO ModBus.MB_Query.Read_Quantity DO
					MB_RegistriHoldingLetti[x+IndirizzoStart] := ModBus.MB_Resp.Data[x];   	(* Vedi tabella *)
				END_FOR

				IndirizzoStart:=254;
				ModBus.MB_Query.Read_StartAddress :=IndirizzoStart - 1 ;
				ModBus.MB_Query.Read_Quantity := 3;
				ModBus.MB_Start := TRUE;

				state := 60;
			END_IF
		END_IF

	60: (* Rispota Altri paramenti *)
		IF NOT ModBus.MB_Start  THEN

			IF ModBus.MB_MASTER.MB_Error<>0 THEN
				state := 300;
			ELSE
				FOR x:=0 TO ModBus.MB_Query.Read_Quantity DO
					MB_RegistriHoldingLetti[x+IndirizzoStart] := ModBus.MB_Resp.Data[x];   	(* Vedi tabella *)
				END_FOR

				WarningAttivoSuCompressore:=MB_RegistriHoldingLetti[255];
				AllarmeAttivoSuCompressore:=MB_RegistriHoldingLetti[256];




				state :=290;
			END_IF
		END_IF


		290:    (* Scrittura il comando di run o stop da remoto*)
		IF NOT ModBus.MB_Start THEN
			IF ModBus.MB_MASTER.MB_Error<>0 THEN (*OR ModBus.MB_MASTER.MB_Error<>0 THEN*)
				state := 300;
			ELSE
				IF AgggiornoStartStop  THEN

					Modbus.MB_Query.FunctionCode := 6;
					Modbus.MB_Query.SlaveAddress := Address;
					ModBus.MB_Query.Write_Quantity :=1;


					IF RUN_REQ THEN
							IndirizzoDaScrivere:=1;
							 DatoDaScrivere:=MB_RegistriHoldingLetti[IndirizzoDaScrivere];
	  							 DatoDaScrivere.0:=TRUE;
  							        DatoDaScrivere.1:=TRUE;
							        DatoDaScrivere.2:=TRUE;
								 RUN_REQ:=FALSE;
					END_IF
					IF STOP_REQ THEN
							IndirizzoDaScrivere:=1;
								 DatoDaScrivere:=MB_RegistriHoldingLetti[IndirizzoDaScrivere];
	  							 DatoDaScrivere.0:=TRUE;
  							        DatoDaScrivere.1:=FALSE;
							        DatoDaScrivere.2:=TRUE;
								 STOP_REQ:=FALSE;
					END_IF
					IF RELEASE_REQ THEN
							IndirizzoDaScrivere:=1;
								 DatoDaScrivere:=MB_RegistriHoldingLetti[IndirizzoDaScrivere];
	  							 DatoDaScrivere.0:=FALSE;
  							        DatoDaScrivere.1:=FALSE;
							        DatoDaScrivere.2:=TRUE;
								 RELEASE_REQ:=FALSE;
					END_IF
			(*		IF CARICO_REQ THEN
								IndirizzoDaScrivere:=1;
							 DatoDaScrivere:=MB_RegistriHoldingLetti[IndirizzoDaScrivere];
	  							 DatoDaScrivere.0:=TRUE;
  							        DatoDaScrivere.1:=TRUE;
							        DatoDaScrivere.2:= NOT DatoDaScrivere.2;
								 CARICO_REQ:=FALSE;
					END_IF  *)

					ModBus.MB_Query.Write_StartAddress := IndirizzoDaScrivere-1;
					ModBus.MB_Query.Write_Data[0] := DatoDaScrivere;
					ModBus.MB_Start := TRUE;
					state := 295;
					AgggiornoStartStop:=FALSE;
				ELSE
					state := 291;
				END_IF
			END_IF
		END_IF


		291:    (* Scrittura BOOL - COIL o WORD *)
		IF NOT ModBus.MB_Start THEN
			IF ModBus.MB_MASTER.MB_Error<>0 THEN (*OR ModBus.MB_MASTER.MB_Error<>0 THEN*)
				state := 300;
			ELSE
				IF LocSelManAuto THEN
					Modbus.MB_Query.FunctionCode := 6;
					Modbus.MB_Query.SlaveAddress := Address;
					ModBus.MB_Query.Write_StartAddress := 112-1;
					ModBus.MB_Query.Write_Quantity :=1;
					ModBus.MB_Query.Write_Data[0] := LocTGP;
					ModBus.MB_Start := TRUE;
					state := 292;
				ELSE
					state := 292;
				END_IF
			END_IF
		END_IF

		292:    (* Scrittura BOOL - COIL o WORD *)
		IF NOT ModBus.MB_Start THEN
			IF ModBus.MB_MASTER.MB_Error<>0 THEN (*OR ModBus.MB_MASTER.MB_Error<>0 THEN*)
				state := 300;
			ELSE
				IF LocSelManAuto THEN
					Modbus.MB_Query.FunctionCode := 6;
					Modbus.MB_Query.SlaveAddress := Address;
					ModBus.MB_Query.Write_StartAddress := 113-1;
					ModBus.MB_Query.Write_Quantity :=1;
					ModBus.MB_Query.Write_Data[0] := LocASP;
					ModBus.MB_Start := TRUE;
					state := 295;
				ELSE
					state := 295;
				END_IF
			END_IF
		END_IF



(*		291:    (* Scrittura BOOL - COIL o WORD *)
		IF NOT ModBus.MB_Start THEN
			IF ModBus.MB_MASTER.MB_Error<>0 THEN (*OR ModBus.MB_MASTER.MB_Error<>0 THEN*)
				state := 300;
			ELSE
				IF ScriviDato THEN
					IF ScriviCoil THEN
						Modbus.MB_Query.FunctionCode := 5;
					ELSE
						Modbus.MB_Query.FunctionCode := 6;
					END_IF
					Modbus.MB_Query.SlaveAddress := Address;
					ModBus.MB_Query.Write_StartAddress := IndirizzoDaScrivere-1;
					ModBus.MB_Query.Write_Quantity :=1;
					ModBus.MB_Query.Write_Data[0] := DatoDaScrivere;
					ModBus.MB_Start := TRUE;
						IF ScriviCoil THEN
							IF 	MB_BitStato[IndirizzoDaScrivere]=WORD_TO_BOOL(DatoDaScrivere-1) THEN
								ScriviDato:=FALSE;
							END_IF
						ELSE
							IF 	MB_RegistriHoldingLetti[IndirizzoDaScrivere]=DatoDaScrivere THEN
								ScriviDato:=FALSE;
							END_IF
						END_IF
					state := 295;
				ELSE
					state := 295;
				END_IF
			END_IF
		END_IF

*)


		295:
		IF NOT ModBus.MB_Start THEN
			IF ModBus.MB_MASTER.MB_Error<>0 THEN (*OR ModBus.MB_MASTER.MB_Error<>0 THEN*)
				state := 300;
			ELSE
				IF fModbusAlr THEN fModbusAlr := FALSE; END_IF
				NodoDaInterrogareCompressoreNuovo:=Address+1;
				InibiscoModbusCompressoreNuovo:=FALSE;
				retryErr := 0;
				retry := 0;
				state := 0;
					IF fModbusAlr=FALSE AND ErroreComuModBus=TRUE THEN
						LogEv(EL_Log,EO_COMPINGRML,ID,62,'ComunicazioneModBus_OK');
						ErroreComuModBus := FALSE;
				(*	WarningCtr := SEL(WarningCtr=0, WarningCtr-1, 0); *)
					END_IF
			END_IF


		END_IF




	(**** CHECK MODBUS ERROR ****)
	300: 	(* Release MODBUS *)
			InibiscoModbusCompressoreNuovo:=FALSE;
			(* Retries *)
			retry:=retry+1;
			IF retry>3 THEN
				retry:=0;

				(* Verify if slave is dead *)
				IF retryErr < retryErrMaX THEN
					retryErr := retryErr + 1;
				ELSE
					fModbusAlr := TRUE;
					(* Verify ModBus error	*)

					IF fModbusAlr AND ErroreComuModBus=FALSE THEN
						LogEv(EL_Alarm,EO_COMPINGRML,ID,61,CONCAT('ErroreModbus_',INT_TO_STRING(ModBus.MB_MASTER.MB_Error)));
						ErroreComuModBus := TRUE;
					END_IF
				END_IF

				END_IF
			Refresh_Now := FALSE;
			NodoDaInterrogareCompressoreNuovo:=Address+1;
			state:=0;
END_CASE




(* Controllo Time Out Ciclo ModBus *)

TimeOutModBus(In:=state<>0,PT:=t#3s);
IF TimeOutModBus.Q THEN
	State:=0;
	Refresh_Now:=TRUE;  (* Rilancio la lettura del nodo *)
	IF MODBUS.MB_Lock=TRUE THEN MODBUS.MB_Lock:=FALSE;END_IF
	IF InibiscoModbusCompressoreNuovo=TRUE THEN InibiscoModbusCompressoreNuovo:=FALSE;END_IF
	NodoDaInterrogareCompressoreNuovo:=Address+1;

END_IF
END_ACTION

(* POU Plant_Objects/obj_MODBUS, ST *)
FUNCTION_BLOCK obj_MODBUS
(* === MODBUS PROTOCOL INTERFACE ===
   v1.1[19/06/15] - Added new VARS allocation and searching
*)
VAR CONSTANT
	VARS_Max	: BYTE := 32;
END_VAR
VAR_INPUT
	(* Settings *)
	ID			: BYTE;
	COM			: BYTE;
	BAUDRATE	: COM_BAUDRATE;
	RS485		: BOOL := FALSE;

	N_STOPBits	:BYTE:=1;

 	(* Interface *)
	MB_MASTER	: MODBUS_EXTENDED_MASTER;
	MB_Start	: BOOL;
	MB_Query	: typModbusExtendedQuery;
	MB_Resp		: typModbusResponse;
	MB_Lock		: BOOL;
	MB_timeOut	: TIME := t#500ms;

	(* Variables management *)
	VARS_En		: BOOL;
	VARS		: ARRAY [0..VARS_Max] OF typ_MODBUS_VAR;
	VARS_Check	: BOOL;
	VARS_Alarm	: BOOL;

	(* Variables allocation *)
	VAR_Pointer : POINTER TO ARRAY[0..99] OF WORD;
	VAR_Cfg		: POINTER TO typ_MODBUS_VAR;
END_VAR
VAR_OUTPUT
	(* Status *)
	Status_Log	: BYTE;
	Status_Vis	: DWORD;
END_VAR
VAR
	sta         : BYTE :=0;
	i			: BYTE;
	j			: BYTE;
	Alarm		: FLT_EVENT;
	
	VarTmr		: TON := (PT:=T#1s);
	VarSta		: BYTE; (* Status *)
	VarCnt		: BYTE; (* Scan counter *)
	VarRetry	: BYTE;
	VarAlarm	: BYTE; (* Last variable with errors *)
END_VAR
IF N_STOPBits=1 THEN MB_MASTER.csCOM_STOPBITS:=STOPBITS_1;END_IF
IF N_STOPBits=2 THEN MB_MASTER.csCOM_STOPBITS:=STOPBITS_2;END_IF

MB_MASTER(ENABLE:=TRUE,	ASCII_Mode:=FALSE, bCOM_PORT:=COM, cbCOM_BAUDRATE:=BAUDRATE, cpCOM_PARITY:=PARITY_NO,
		cbsCOM_BYTESIZE:=BS_8, cfCOM_FLOW_CONTROL:=SEL(RS485,NO_FLOW_CONTROL,HALFDUPLEX),
		tTIME_OUT:=MB_timeOut,	StartFunction:=MB_Start, ExtQuery:=MB_Query, Response:=MB_Resp);

(* Process variable management *)
IF VARS_En THEN VARS_Process(); END_IF

(* Check status *)
Alarm(IN:=(MB_MASTER.bInterfaceError<>0));
IF Alarm.EVH THEN
	LogEv(SEL(MB_MASTER.bInterfaceError<>3,EL_Wrn,EL_Alarm),EO_MODBUS,ID,1,BYTE_TO_STRING(MB_MASTER.bInterfaceError));
END_IF
IF Alarm.EVL THEN								(* Trigger a fall edge: MODBUS back working *)
	LogEv(EL_Log,EO_MODBUS,ID,2,'MODBUS_OK');
END_IF

(* Log/visu status *)
   IF Alarm.IN   THEN Status_Log:=2; Status_Vis:=COLOR_RED;
ELSIF Vars_Alarm THEN Status_Log:=1; Status_Vis:=COLOR_YELLOW;
  				 ELSE Status_Log:=0; Status_Vis:=COLOR_GREEN;
END_IF
END_FUNCTION_BLOCK
ACTION VAR_Search:
(* Search VAR with specific pointer if not found return first free VAR
	[Last VAR is not active... used as safe area...] 
*)
j:=VARS_Max;
FOR i := 0 TO VARS_Max-1 DO
	IF VARS[i].Variable=0 AND j>i THEN j:=i; END_IF
	IF VARS[i].Variable=VAR_Pointer THEN
		VAR_Cfg:=ADR(VARS[i]);
		RETURN;
	END_IF
END_FOR
VAR_Cfg:=ADR(VARS[j]);
END_ACTION
ACTION VARS_Process:
(* Update var timers *)
VarTmr(IN:=(NOT VarTmr.Q));
IF VarTmr.Q THEN
	FOR i := 0 TO VARS_Max DO
		IF VARS[i].Refresh_Cnt>0 THEN VARS[i].Refresh_Cnt:=VARS[i].Refresh_Cnt-1; END_IF
	END_FOR
	VARS_Check:=TRUE;
END_IF


(* Process status *)
CASE VarSta OF
	0: (* === Init *)
		VarCnt:=0;
		VarSta:=1;

	1: (* === Wait check signal *)
		IF VARS_Check THEN				(* Decremented "Refresh_Cnt" *)
			VARS_Check:=FALSE;
			VarCnt:=0;
			VarSta:=2;
		END_IF

